DATA_BLOCK "DB_CrossCut_Opt_HMI"
{ DB_Accessible_From_OPC_UA := 'FALSE' ;
 DB_Accessible_From_Webserver := 'FALSE' ;
 S7_Optimized_Access := 'FALSE' }
VERSION : 0.1
NON_RETAIN
   STRUCT
      tALM { ExternalWritable := 'False'} : Struct   // HMI Alarms
         tE { ExternalWritable := 'False'} : Struct   // Stopping faults
            xSpare_0 { ExternalWritable := 'False'} : Bool;
            xSpare_1 { ExternalWritable := 'False'} : Bool;
            xSpare_2 { ExternalWritable := 'False'} : Bool;
            xSpare_3 { ExternalWritable := 'False'} : Bool;
            xSpare_4 { ExternalWritable := 'False'} : Bool;
            xSpare_5 { ExternalWritable := 'False'} : Bool;
            xSpare_6 { ExternalWritable := 'False'} : Bool;
            xSpare_7 { ExternalWritable := 'False'} : Bool;
            xSpare_8 { ExternalWritable := 'False'} : Bool;
            xSpare_9 { ExternalWritable := 'False'} : Bool;
            xSpare_10 { ExternalWritable := 'False'} : Bool;
            xSpare_11 { ExternalWritable := 'False'} : Bool;
            xSpare_12 { ExternalWritable := 'False'} : Bool;
            xSpare_13 { ExternalWritable := 'False'} : Bool;
            xSpare_14 { ExternalWritable := 'False'} : Bool;
            xSpare_15 { ExternalWritable := 'False'} : Bool;
            xSpare_16 { ExternalWritable := 'False'} : Bool;
            xSpare_17 { ExternalWritable := 'False'} : Bool;
            xSpare_18 { ExternalWritable := 'False'} : Bool;
            xSpare_19 { ExternalWritable := 'False'} : Bool;
            xSpare_20 { ExternalWritable := 'False'} : Bool;
            xSpare_21 { ExternalWritable := 'False'} : Bool;
            xSpare_22 { ExternalWritable := 'False'} : Bool;
            xSpare_23 { ExternalWritable := 'False'} : Bool;
            xSpare_24 { ExternalWritable := 'False'} : Bool;
            xSpare_25 { ExternalWritable := 'False'} : Bool;
            xSpare_26 { ExternalWritable := 'False'} : Bool;
            xSpare_27 { ExternalWritable := 'False'} : Bool;
            xSpare_28 { ExternalWritable := 'False'} : Bool;
            xSpare_29 { ExternalWritable := 'False'} : Bool;
            xSpare_30 { ExternalWritable := 'False'} : Bool;
            xSpare_31 { ExternalWritable := 'False'} : Bool;
         END_STRUCT;
         tS { ExternalWritable := 'False'} : Struct   // Stopping faults
            xSpare_0 { ExternalWritable := 'False'} : Bool;
            xSpare_1 { ExternalWritable := 'False'} : Bool;
            xSpare_2 { ExternalWritable := 'False'} : Bool;
            xSpare_3 { ExternalWritable := 'False'} : Bool;
            xSpare_4 { ExternalWritable := 'False'} : Bool;
            xSpare_5 { ExternalWritable := 'False'} : Bool;
            xSpare_6 { ExternalWritable := 'False'} : Bool;
            xSpare_7 { ExternalWritable := 'False'} : Bool;
            xSpare_8 { ExternalWritable := 'False'} : Bool;
            xSpare_9 { ExternalWritable := 'False'} : Bool;
            xSpare_10 { ExternalWritable := 'False'} : Bool;
            xSpare_11 { ExternalWritable := 'False'} : Bool;
            xSpare_12 { ExternalWritable := 'False'} : Bool;
            xSpare_13 { ExternalWritable := 'False'} : Bool;
            xSpare_14 { ExternalWritable := 'False'} : Bool;
            xSpare_15 { ExternalWritable := 'False'} : Bool;
            xSpare_16 { ExternalWritable := 'False'} : Bool;
            xSpare_17 { ExternalWritable := 'False'} : Bool;
            xSpare_18 { ExternalWritable := 'False'} : Bool;
            xSpare_19 { ExternalWritable := 'False'} : Bool;
            xSpare_20 { ExternalWritable := 'False'} : Bool;
            xSpare_21 { ExternalWritable := 'False'} : Bool;
            xSpare_22 { ExternalWritable := 'False'} : Bool;
            xSpare_23 { ExternalWritable := 'False'} : Bool;
            xSpare_24 { ExternalWritable := 'False'} : Bool;
            xSpare_25 { ExternalWritable := 'False'} : Bool;
            xSpare_26 { ExternalWritable := 'False'} : Bool;
            xSpare_27 { ExternalWritable := 'False'} : Bool;
            xSpare_28 { ExternalWritable := 'False'} : Bool;
            xSpare_29 { ExternalWritable := 'False'} : Bool;
            xSpare_30 { ExternalWritable := 'False'} : Bool;
            xSpare_31 { ExternalWritable := 'False'} : Bool;
         END_STRUCT;
         tF { ExternalWritable := 'False'} : Struct   // Faults
            xSpare_0 { ExternalWritable := 'False'} : Bool;
            xSpare_1 { ExternalWritable := 'False'} : Bool;
            xSpare_2 { ExternalWritable := 'False'} : Bool;
            xSpare_3 { ExternalWritable := 'False'} : Bool;
            xSpare_4 { ExternalWritable := 'False'} : Bool;
            xSpare_5 { ExternalWritable := 'False'} : Bool;
            xSpare_6 { ExternalWritable := 'False'} : Bool;
            xSpare_7 { ExternalWritable := 'False'} : Bool;
            xSpare_8 { ExternalWritable := 'False'} : Bool;
            xSpare_9 { ExternalWritable := 'False'} : Bool;
            xSpare_10 { ExternalWritable := 'False'} : Bool;
            xSpare_11 { ExternalWritable := 'False'} : Bool;
            xSpare_12 { ExternalWritable := 'False'} : Bool;
            xSpare_13 { ExternalWritable := 'False'} : Bool;
            xSpare_14 { ExternalWritable := 'False'} : Bool;
            xSpare_15 { ExternalWritable := 'False'} : Bool;
            xSpare_16 { ExternalWritable := 'False'} : Bool;
            xSpare_17 { ExternalWritable := 'False'} : Bool;
            xSpare_18 { ExternalWritable := 'False'} : Bool;
            xSpare_19 { ExternalWritable := 'False'} : Bool;
            xSpare_20 { ExternalWritable := 'False'} : Bool;
            xSpare_21 { ExternalWritable := 'False'} : Bool;
            xSpare_22 { ExternalWritable := 'False'} : Bool;
            xSpare_23 { ExternalWritable := 'False'} : Bool;
            xSpare_24 { ExternalWritable := 'False'} : Bool;
            xSpare_25 { ExternalWritable := 'False'} : Bool;
            xSpare_26 { ExternalWritable := 'False'} : Bool;
            xSpare_27 { ExternalWritable := 'False'} : Bool;
            xSpare_28 { ExternalWritable := 'False'} : Bool;
            xSpare_29 { ExternalWritable := 'False'} : Bool;
            xSpare_30 { ExternalWritable := 'False'} : Bool;
            xSpare_31 { ExternalWritable := 'False'} : Bool;
         END_STRUCT;
         tW { ExternalWritable := 'False'} : Struct   // Warnings
            xSpare_0 { ExternalWritable := 'False'} : Bool;
            xSpare_1 { ExternalWritable := 'False'} : Bool;
            xSpare_2 { ExternalWritable := 'False'} : Bool;
            xSpare_3 { ExternalWritable := 'False'} : Bool;
            xSpare_4 { ExternalWritable := 'False'} : Bool;
            xSpare_5 { ExternalWritable := 'False'} : Bool;
            xSpare_6 { ExternalWritable := 'False'} : Bool;
            xSpare_7 { ExternalWritable := 'False'} : Bool;
            xSpare_8 { ExternalWritable := 'False'} : Bool;
            xSpare_9 { ExternalWritable := 'False'} : Bool;
            xSpare_10 { ExternalWritable := 'False'} : Bool;
            xSpare_11 { ExternalWritable := 'False'} : Bool;
            xSpare_12 { ExternalWritable := 'False'} : Bool;
            xSpare_13 { ExternalWritable := 'False'} : Bool;
            xSpare_14 { ExternalWritable := 'False'} : Bool;
            xSpare_15 { ExternalWritable := 'False'} : Bool;
            xSpare_16 { ExternalWritable := 'False'} : Bool;
            xSpare_17 { ExternalWritable := 'False'} : Bool;
            xSpare_18 { ExternalWritable := 'False'} : Bool;
            xSpare_19 { ExternalWritable := 'False'} : Bool;
            xSpare_20 { ExternalWritable := 'False'} : Bool;
            xSpare_21 { ExternalWritable := 'False'} : Bool;
            xSpare_22 { ExternalWritable := 'False'} : Bool;
            xSpare_23 { ExternalWritable := 'False'} : Bool;
            xSpare_24 { ExternalWritable := 'False'} : Bool;
            xSpare_25 { ExternalWritable := 'False'} : Bool;
            xSpare_26 { ExternalWritable := 'False'} : Bool;
            xSpare_27 { ExternalWritable := 'False'} : Bool;
            xSpare_28 { ExternalWritable := 'False'} : Bool;
            xSpare_29 { ExternalWritable := 'False'} : Bool;
            xSpare_30 { ExternalWritable := 'False'} : Bool;
            xSpare_31 { ExternalWritable := 'False'} : Bool;
         END_STRUCT;
      END_STRUCT;
      tHMR { ExternalWritable := 'False'} : Struct   // HMI Read
         xEnabledPriority { ExternalWritable := 'False'} : Bool;   // Enabled/disable priority (1=enabled) {X|X|X|X|O}
         xSpare1 { ExternalWritable := 'False'} : Bool;
         xSpare2 { ExternalWritable := 'False'} : Bool;
         xSpare3 { ExternalWritable := 'False'} : Bool;
         xSpare4 { ExternalWritable := 'False'} : Bool;
         xSpare5 { ExternalWritable := 'False'} : Bool;
         xSpare6 { ExternalWritable := 'False'} : Bool;
         xSpare7 { ExternalWritable := 'False'} : Bool;
         xSpare8 { ExternalWritable := 'False'} : Bool;
         xSpare9 { ExternalWritable := 'False'} : Bool;
         xSpare10 { ExternalWritable := 'False'} : Bool;
         xSpare11 { ExternalWritable := 'False'} : Bool;
         xSpare12 { ExternalWritable := 'False'} : Bool;
         xSpare13 { ExternalWritable := 'False'} : Bool;
         xSpare14 { ExternalWritable := 'False'} : Bool;   //
         xSpare15 { ExternalWritable := 'False'} : Bool;
         xSpare16 { ExternalWritable := 'False'} : Bool;
         xSpare17 { ExternalWritable := 'False'} : Bool;
         xSpare18 { ExternalWritable := 'False'} : Bool;
         xSpare19 { ExternalWritable := 'False'} : Bool;
         xSpare20 { ExternalWritable := 'False'} : Bool;
         xSpare21 { ExternalWritable := 'False'} : Bool;
         xSpare22 { ExternalWritable := 'False'} : Bool;
         xSpare23 { ExternalWritable := 'False'} : Bool;
         xSpare24 { ExternalWritable := 'False'} : Bool;
         xSpare25 { ExternalWritable := 'False'} : Bool;
         xSpare26 { ExternalWritable := 'False'} : Bool;
         xSpare27 { ExternalWritable := 'False'} : Bool;
         xSpare28 { ExternalWritable := 'False'} : Bool;
         xSpare29 { ExternalWritable := 'False'} : Bool;
         xSpare30 { ExternalWritable := 'False'} : Bool;
         xSpare31 { ExternalWritable := 'False'} : Bool;
         xSpare { ExternalWritable := 'False'} : Array[0..15] of Bool;
         iSpare0 { ExternalWritable := 'False'} : Int;
         iSpare1 { ExternalWritable := 'False'} : Int;
         iSpare2 { ExternalWritable := 'False'} : Int;
         iSpare3 { ExternalWritable := 'False'} : Int;
         iSpare4 { ExternalWritable := 'False'} : Int;
         iSpare5 { ExternalWritable := 'False'} : Int;
         iSpare6 { ExternalWritable := 'False'} : Int;
         iSpare7 { ExternalWritable := 'False'} : Int;
         iSpare8 { ExternalWritable := 'False'} : Int;
         iSpare9 { ExternalWritable := 'False'} : Int;
         iSpare10 { ExternalWritable := 'False'} : Int;
         iSpare11 { ExternalWritable := 'False'} : Int;
         iSpare12 { ExternalWritable := 'False'} : Int;
         iSpare13 { ExternalWritable := 'False'} : Int;
         iSpare14 { ExternalWritable := 'False'} : Int;
         iSpare15 { ExternalWritable := 'False'} : Int;
         iSpare16 { ExternalWritable := 'False'} : Int;
         dSpare0 { ExternalWritable := 'False'} : DInt;   //
         dSpare1 { ExternalWritable := 'False'} : DInt;   //
         dSpare2 { ExternalWritable := 'False'} : DInt;
         dSpare3 { ExternalWritable := 'False'} : DInt;
         dSpare4 { ExternalWritable := 'False'} : DInt;
         dSpare5 { ExternalWritable := 'False'} : DInt;
         dSpare6 { ExternalWritable := 'False'} : DInt;
         dSpare7 { ExternalWritable := 'False'} : DInt;
         dSpare8 { ExternalWritable := 'False'} : DInt;
         dSpare9 { ExternalWritable := 'False'} : DInt;
         dSpare10 { ExternalWritable := 'False'} : DInt;
         dSpare11 { ExternalWritable := 'False'} : DInt;
         dSpare12 { ExternalWritable := 'False'} : DInt;
         dSpare13 { ExternalWritable := 'False'} : DInt;
         dSpare14 { ExternalWritable := 'False'} : DInt;
         dSpare15 { ExternalWritable := 'False'} : DInt;
         rSpare0 { ExternalWritable := 'False'} : Real;
         rSpare1 { ExternalWritable := 'False'} : Real;
         rSpare2 { ExternalWritable := 'False'} : Real;
         rSpare3 { ExternalWritable := 'False'} : Real;
         rSpare4 { ExternalWritable := 'False'} : Real;
         rSpare5 { ExternalWritable := 'False'} : Real;
         rSpare6 { ExternalWritable := 'False'} : Real;
         rSpare7 { ExternalWritable := 'False'} : Real;
         rSpare8 { ExternalWritable := 'False'} : Real;
         tManCmd { ExternalWritable := 'False'} : Struct
            xSpare0 { ExternalWritable := 'False'} : Bool;   //
            xSpare1 { ExternalWritable := 'False'} : Bool;
            xSpare2 { ExternalWritable := 'False'} : Bool;
            xSpare3 { ExternalWritable := 'False'} : Bool;
            xSpare4 { ExternalWritable := 'False'} : Bool;
            xSpare5 { ExternalWritable := 'False'} : Bool;
            xSpare6 { ExternalWritable := 'False'} : Bool;
            xSpare7 { ExternalWritable := 'False'} : Bool;
            xSpare8 { ExternalWritable := 'False'} : Bool;
            xSpare9 { ExternalWritable := 'False'} : Bool;
            xSpare10 { ExternalWritable := 'False'} : Bool;
            xSpare11 { ExternalWritable := 'False'} : Bool;
            xSpare12 { ExternalWritable := 'False'} : Bool;
            xSpare13 { ExternalWritable := 'False'} : Bool;
            xSpare14 { ExternalWritable := 'False'} : Bool;
            xSpare15 { ExternalWritable := 'False'} : Bool;
            xSpare { ExternalWritable := 'False'} : Array[0..15] of Bool;
         END_STRUCT;
      END_STRUCT;
      tHMW : Struct   // HMI Write
         xEnDisPriority : Bool;   // Enable/disable priority (1=enabled) {X|X|X|X|O}
         xSpare1 : Bool;
         xSpare2 : Bool;
         xSpare3 : Bool;
         xSpare4 : Bool;
         xSpare5 : Bool;
         xSpare6 : Bool;
         xSpare7 : Bool;
         xSpare8 : Bool;
         xSpare9 : Bool;
         xSpare10 : Bool;   //
         xSpare11 : Bool;
         xSpare12 : Bool;
         xSpare13 : Bool;
         xSpare14 : Bool;   //
         xSpare15 : Bool;
         xSpare16 : Bool;
         xSpare17 : Bool;
         xSpare18 : Bool;
         xSpare19 : Bool;
         xSpare20 : Bool;
         xSpare21 : Bool;
         xSpare22 : Bool;
         xSpare23 : Bool;
         xSpare24 : Bool;
         xSpare25 : Bool;
         xSpare26 : Bool;
         xSpare27 : Bool;
         xSpare28 : Bool;
         xSpare29 : Bool;
         xSpare30 : Bool;
         xSpare31 : Bool;
         xSpare : Array[0..15] of Bool;
         iSpare0 : Int;
         iSpare1 : Int;
         iSpare2 : Int;
         iSpare3 : Int;
         iSpare4 : Int;
         iSpare5 : Int;
         iSpare6 : Int;
         iSpare7 : Int;
         iSpare8 : Int;
         iSpare9 : Int;
         iSpare10 : Int;
         iSpare11 : Int;
         iSpare12 : Int;
         iSpare13 : Int;
         iSpare14 : Int;
         iSpare15 : Int;
         iSpare16 : Int;
         dSpare0 : DInt;   //
         dSpare1 : Int;   //
         dSpare2 : Int;   //
         dSpare3 : DInt;
         dSpare4 : DInt;
         dSpare5 : DInt;
         dSpare6 : DInt;
         dSpare7 : DInt;
         dSpare8 : DInt;
         dSpare9 : DInt;
         dSpare10 : DInt;
         dSpare11 : DInt;
         dSpare12 : DInt;
         dSpare13 : DInt;
         dSpare14 : DInt;
         dSpare15 : DInt;
         dSpare16 : DInt;
         rSpare0 : Real;
         rSpare1 : Real;
         rSpare2 : Real;
         rSpare3 : Real;
         rSpare4 : Real;
         rSpare5 : Real;
         rSpare6 : Real;
         rSpare7 : Real;
         rSpare8 : Real;
         tManCmd : Struct
            xSpare0 : Bool;   //
            xSpare1 : Bool;
            xSpare2 { ExternalWritable := 'False'} : Bool;
            xSpare3 { ExternalWritable := 'False'} : Bool;
            xSpare4 { ExternalWritable := 'False'} : Bool;
            xSpare5 { ExternalWritable := 'False'} : Bool;
            xSpare6 { ExternalWritable := 'False'} : Bool;
            xSpare7 { ExternalWritable := 'False'} : Bool;
            xSpare8 { ExternalWritable := 'False'} : Bool;
            xSpare9 { ExternalWritable := 'False'} : Bool;
            xSpare10 { ExternalWritable := 'False'} : Bool;
            xSpare11 { ExternalWritable := 'False'} : Bool;
            xSpare12 { ExternalWritable := 'False'} : Bool;
            xSpare13 { ExternalWritable := 'False'} : Bool;
            xSpare14 { ExternalWritable := 'False'} : Bool;
            xSpare15 { ExternalWritable := 'False'} : Bool;
            xSpare16 : Bool;
            xSpare17 : Bool;
            xSpare18 : Bool;
            xSpare19 : Bool;
            xSpare20 : Bool;
            xSpare21 : Bool;
            xSpare22 : Bool;
            xSpare23 : Bool;
            xSpare24 : Bool;
            xSpare25 : Bool;
            xSpare26 : Bool;
            xSpare27 : Bool;
            xSpare28 : Bool;
            xSpare29 : Bool;
            xSpare30 : Bool;
            xSpare31 : Bool;
         END_STRUCT;
      END_STRUCT;
   END_STRUCT;


BEGIN

END_DATA_BLOCK

DATA_BLOCK "DB_CrossCut_1_HMI"
{ DB_Accessible_From_OPC_UA := 'FALSE' ;
 DB_Accessible_From_Webserver := 'FALSE' ;
 S7_Optimized_Access := 'FALSE' }
VERSION : 0.1
NON_RETAIN
   STRUCT
      tALM : Struct   // HMI Alarms
         tE : Struct   // Emergency alarms
            xLocON : Bool;   // KE.Local emergency ON {X|X|X|X|O}
            xLocal1 : Bool;   // SB.Local emergency push button 1 {X|X|X|X|O}
            xLocal2 : Bool;   // SB.Local emergency push button 2 {X|X|X|X|O}
            xLocal3 : Bool;   // SB.Local emergency push button 3 {X|X|X|X|O}
            xSpare_4 : Bool;
            xSpare_5 : Bool;
            xSpare_6 : Bool;
            xSpare_7 : Bool;
            xSpare_8 : Bool;
            xSpare_9 : Bool;
            xSpare_10 : Bool;
            xSpare_11 : Bool;
            xSpare_12 : Bool;
            xSpare_13 : Bool;
            xSpare_14 : Bool;
            xSpare_15 : Bool;
            xSpare_16 : Bool;
            xSpare_17 : Bool;
            xSpare_18 : Bool;
            xSpare_19 : Bool;
            xSpare_20 : Bool;
            xSpare_21 : Bool;
            xSpare_22 : Bool;
            xSpare_23 : Bool;
            xSpare_24 : Bool;
            xSpare_25 : Bool;
            xSpare_26 : Bool;
            xSpare_27 : Bool;
            xSpare_28 : Bool;
            xSpare_29 : Bool;
            xSpare_30 : Bool;
            xSpare_31 : Bool;
         END_STRUCT;
         tS : Struct   // Stopping faults
            xAxisNotAvail : Bool;   // AZ.Axis not available {X|X|X|X|O}
            xInpInstallation : Bool;   // L+.Input power supply ON {X|X|X|X|O}
            xAuxPower : Bool;   // L+.Auxiliary power supple set-in {X|X|X|X|O}
            xAreaSafety : Bool;   // KE.Area safety {X|X|X|X|O}
            xOverstroke : Bool;   // KA.Carriage overstroke {X|X|X|X|O}
            xExternInputPower : Bool;   // L+.External input power supply {X|X|X|X|O}
            xCarriageCutOut : Bool;   // QM.Carriage translation overload {X|X|X|X|O}
            xDriveTrip : Bool;   // AZ.Drive trip {X|X|X|X|O}
            xDriveNotEnabled : Bool;   // AZ.Drive not enabled {X|X|X|X|O}
            xAxisNotReady : Bool;   // AZ.Axis not ready {X|X|X|X|O}
            xDriveNotReady : Bool;   // AZ.Drive not ready {X|X|X|X|O}
            xAxisNotSyncro : Bool;   // AZ.Axis not syncronized {X|X|X|X|O}
            xSpare_12 : Bool;
            xSpare_13 : Bool;
            xSpare_14 : Bool;
            xSpare_15 : Bool;
            xSpare_16 : Bool;
            xSpare_17 : Bool;
            xSpare_18 : Bool;
            xSpare_19 : Bool;
            xSpare_20 : Bool;
            xSpare_21 : Bool;
            xSpare_22 : Bool;
            xSpare_23 : Bool;
            xSpare_24 : Bool;
            xSpare_25 : Bool;
            xSpare_26 : Bool;
            xSpare_27 : Bool;
            xSpare_28 : Bool;
            xSpare_29 : Bool;
            xSpare_30 : Bool;
            xSpare_31 : Bool;
         END_STRUCT;
         tF : Struct   // Faults
            xSpare_0 : Bool;
            xSpare_1 : Bool;
            xSpare_2 : Bool;
            xSpare_3 : Bool;
            xSpare_4 : Bool;
            xSpare_5 : Bool;
            xSpare_6 : Bool;
            xSpare_7 : Bool;
            xSpare_8 : Bool;
            xSpare_9 : Bool;
            xSpare_10 : Bool;
            xSpare_11 : Bool;
            xSpare_12 : Bool;
            xSpare_13 : Bool;
            xSpare_14 : Bool;
            xSpare_15 : Bool;
            xSpare_16 : Bool;
            xSpare_17 : Bool;
            xSpare_18 : Bool;
            xSpare_19 : Bool;
            xSpare_20 : Bool;
            xSpare_21 : Bool;
            xSpare_22 : Bool;
            xSpare_23 : Bool;
            xSpare_24 : Bool;
            xSpare_25 : Bool;
            xSpare_26 : Bool;
            xSpare_27 : Bool;
            xSpare_28 : Bool;
            xSpare_29 : Bool;
            xSpare_30 : Bool;
            xSpare_31 : Bool;
         END_STRUCT;
         tW : Struct   // Warnings
            xSpare_0 : Bool;
            xSpare_1 : Bool;
            xSpare_2 : Bool;
            xSpare_3 : Bool;
            xSpare_4 : Bool;
            xSpare_5 : Bool;
            xSpare_6 : Bool;
            xSpare_7 : Bool;
            xSpare_8 : Bool;
            xSpare_9 : Bool;
            xSpare_10 : Bool;
            xSpare_11 : Bool;
            xSpare_12 : Bool;
            xSpare_13 : Bool;
            xSpare_14 : Bool;
            xSpare_15 : Bool;
            xSpare_16 : Bool;
            xSpare_17 : Bool;
            xSpare_18 : Bool;
            xSpare_19 : Bool;
            xSpare_20 : Bool;
            xSpare_21 : Bool;
            xSpare_22 : Bool;
            xSpare_23 : Bool;
            xSpare_24 : Bool;
            xSpare_25 : Bool;
            xSpare_26 : Bool;
            xSpare_27 : Bool;
            xSpare_28 : Bool;
            xSpare_29 : Bool;
            xSpare_30 : Bool;
            xSpare_31 : Bool;
         END_STRUCT;
      END_STRUCT;
      tHMR : Struct   // HMI Read
         xSpare0 : Bool;   //
         xSpare1 : Bool;   //
         xSpare2 : Bool;
         xSpare3 : Bool;
         xSpare4 : Bool;
         xSpare5 : Bool;
         xSpare6 : Bool;
         xSpare7 : Bool;
         xSpare8 : Bool;
         xSpare9 : Bool;
         xSpare10 : Bool;
         xSpare11 : Bool;
         xSpare12 : Bool;
         xSpare13 : Bool;
         xManualCommandEnabled : Bool;   // Manual Command enabled {x|x|x|x|O}
         xSpare15 : Bool;
         xSpare16 : Bool;
         xSpare17 : Bool;
         xSpare18 : Bool;
         xSpare19 : Bool;
         xSpare20 : Bool;
         xSpare21 : Bool;
         xSpare22 : Bool;
         xSpare23 : Bool;
         xSpare24 : Bool;
         xSpare25 : Bool;
         xSpare26 : Bool;
         xSpare27 : Bool;
         xSpare28 : Bool;
         xSpare29 : Bool;
         xSpare30 : Bool;
         xSpare31 : Bool;
         xSpare : Array[0..15] of Bool;
         iSpare0 { ExternalWritable := 'False'} : Int;
         iSpare1 { ExternalWritable := 'False'} : Int;
         iSpare2 { ExternalWritable := 'False'} : Int;
         iSpare3 { ExternalWritable := 'False'} : Int;
         iSpare4 { ExternalWritable := 'False'} : Int;
         iSpare5 { ExternalWritable := 'False'} : Int;
         iSpare6 { ExternalWritable := 'False'} : Int;
         iSpare7 { ExternalWritable := 'False'} : Int;
         iSpare8 { ExternalWritable := 'False'} : Int;
         iSpare9 { ExternalWritable := 'False'} : Int;
         iSpare10 { ExternalWritable := 'False'} : Int;
         iSpare11 { ExternalWritable := 'False'} : Int;
         iSpare12 { ExternalWritable := 'False'} : Int;
         iSpare13 { ExternalWritable := 'False'} : Int;
         iSpare14 { ExternalWritable := 'False'} : Int;
         iSpare15 { ExternalWritable := 'False'} : Int;
         iSpare16 { ExternalWritable := 'False'} : Int;
         dDistanceSnaproll_cmm { ExternalWritable := 'False'} : DInt;   // Distance from snaproll [mm/100] {mm/100|mm|x|x|M}
         dStatus { ExternalWritable := 'False'} : DInt;   // XCut actual status (1=Idle 3=Running 7=Faulted)  {X|X|X|X|O}
         dXCutActualStatus { ExternalWritable := 'False'} : DInt;   // XCut actual status (1=Disabled 3=Enabled) {X|X|X|X|O}
         dXCutStatusRequest { ExternalWritable := 'False'} : DInt;   // XCut status request (1=Disabled 3=Enabled) {X|X|X|X|O}
         dDistanceFromCenterLine_cmm { ExternalWritable := 'False'} : DInt;   // Distance from center line [mm/100] {mm/100|mm|X|X|O}
         dAngleValue_uDegree { ExternalWritable := 'False'} : DInt;   // Angle value [°/1000000] {°/1000000|°|X|X|O}
         dActualCutPosRequest { ExternalWritable := 'False'} : DInt;   // Actual cut position request (1=By operator 2=On gross ribbon 3=On net ribbon 4=On YCut position) {X|X|X|X|O}
         dCarriagePosition_cmm { ExternalWritable := 'False'} : DInt;   // Actual carriage position [mm/100]
         dSpare8 { ExternalWritable := 'False'} : DInt;
         dSpare9 { ExternalWritable := 'False'} : DInt;
         dSpare10 { ExternalWritable := 'False'} : DInt;
         dSpare11 { ExternalWritable := 'False'} : DInt;
         dSpare12 { ExternalWritable := 'False'} : DInt;
         dSpare13 { ExternalWritable := 'False'} : DInt;
         dSpare14 { ExternalWritable := 'False'} : DInt;
         dSpare15 { ExternalWritable := 'False'} : DInt;
         rHeadUsage_km { ExternalWritable := 'False'} : Real;   // Head usage [Km] {Km|Km|X|X|O}
         rSpare1 { ExternalWritable := 'False'} : Real;
         rSpare2 { ExternalWritable := 'False'} : Real;
         rSpare3 { ExternalWritable := 'False'} : Real;
         rSpare4 { ExternalWritable := 'False'} : Real;
         rSpare5 { ExternalWritable := 'False'} : Real;
         rSpare6 { ExternalWritable := 'False'} : Real;
         rSpare7 { ExternalWritable := 'False'} : Real;
         rSpare8 { ExternalWritable := 'False'} : Real;
         tManCmd { ExternalWritable := 'False'} : Struct
            xManJogFwdFdbk { ExternalWritable := 'False'} : Bool;   // Manual jog forward feedback {X|X|X|X|O}
            xManJogBckFdbk { ExternalWritable := 'False'} : Bool;   // Manual jog backward feedback {X|X|X|X|O}
            xManCarriageDownFdbk { ExternalWritable := 'False'} : Bool;   // Manual carriage down feedback {X|X|X|X|O}
            xManFireONFdbk { ExternalWritable := 'False'} : Bool;   // Manual fire ON feedback {X|X|X|X|O}
            xManOilONFdbk { ExternalWritable := 'False'} : Bool;   // Manual oil ON feedback {X|X|X|X|O}
            xSpare5 { ExternalWritable := 'False'} : Bool;
            xSpare6 { ExternalWritable := 'False'} : Bool;
            xSpare7 { ExternalWritable := 'False'} : Bool;
            xSpare8 { ExternalWritable := 'False'} : Bool;
            xSpare9 { ExternalWritable := 'False'} : Bool;
            xSpare10 { ExternalWritable := 'False'} : Bool;
            xSpare11 { ExternalWritable := 'False'} : Bool;
            xSpare12 { ExternalWritable := 'False'} : Bool;
            xSpare13 { ExternalWritable := 'False'} : Bool;
            xSpare14 { ExternalWritable := 'False'} : Bool;
            xSpare15 { ExternalWritable := 'False'} : Bool;
            xSpare { ExternalWritable := 'False'} : Array[0..15] of Bool;
         END_STRUCT;
      END_STRUCT;
      tHMW : Struct   // HMI Write
         xCutBreakEnabled { ExternalWritable := 'False'} : Bool;   // Cut on glass break enabled {X|X|X|X|O}
         xIncAngleValue : Bool;   // Increment angle value {X|X|X|X|O}
         xDecAngleValue : Bool;   // Decrement angle value {X|X|X|X|O}
         xCalibDistRequest : Bool;   // Calibration distance request {X|X|X|X|O}
         xCalibDiagRequest : Bool;   // Calibration diagonal request {X|X|X|X|O}
         xCutOperator : Bool;   // Cutting position by operator request {X|X|X|X|O}
         xCutGross : Bool;   // Cutting position by gross width position {X|X|X|X|O}
         xCutNet : Bool;   // Cutting position by net width position {X|X|X|X|O}
         xCutYCut : Bool;   // Cutting position by YCut position {X|X|X|X|O}
         xSpare9 : Bool;
         xSpare10 : Bool;
         xSpare11 : Bool;
         xSpare12 : Bool;
         xResetHeadUsage : Bool;   // Reset the head usage {X|X|X|X|O}
         xEnableManualCommand : Bool;   // Enable Disable Manual command {x|x|x|x|O}
         xUpdateDistanceSnaproll : Bool;   // Update distance from snaproll {x|x|x|x|M}
         xUpdateDistCenterLine : Bool;   // Update distance from center line {X|X|X|X|M}
         xUpdateAngleValue : Bool;   // Update angle value {X|X|X|X|M}
         xSpare18 : Bool;
         xSpare19 : Bool;
         xSpare20 : Bool;
         xSpare21 : Bool;
         xSpare22 : Bool;
         xSpare23 : Bool;
         xSpare24 : Bool;
         xSpare25 : Bool;
         xSpare26 : Bool;
         xSpare27 : Bool;
         xSpare28 : Bool;
         xSpare29 : Bool;
         xSpare30 : Bool;
         xSpare31 : Bool;
         xSpare : Array[0..15] of Bool;
         iSpare0 : Int;
         iSpare1 : Int;
         iSpare2 : Int;
         iSpare3 : Int;
         iSpare4 : Int;
         iSpare5 : Int;
         iSpare6 : Int;
         iSpare7 : Int;
         iSpare8 : Int;
         iSpare9 : Int;
         iSpare10 : Int;
         iSpare11 : Int;
         iSpare12 : Int;
         iSpare13 : Int;
         iSpare14 : Int;
         iSpare15 : Int;
         iSpare16 : Int;
         dDistanceSnaproll_cmm : DInt;   // Distance from snaproll [mm/100] {mm/100|mm|1|70000|M}
         dDistanceFromCenterLine_cmm : DInt;   // Distance from center line [mm/100] {mm/100|mm|-3000|0|M}
         dAngleValue_uDegree : DInt;   // Bridge angle value [°/1000000] {°/1000000|°|7|9|M}
         dOperStartCutPos_cmm : DInt;   // Operator start cut position [mm/100] {mm/100|mm|-3000|0|O}
         dOperEndCutPos_cmm : DInt;   // Operator end cut position  [mm/100] {mm/100|mm|0|3000|O}
         dDescReactTime_ms : DInt;   // Carriage descent reaction time [ms] {ms|s|0|1|M}
         dRaiseReactTime_ms : DInt;   // Carriage raise reaction time [ms] {ms|s|0|1|M}
         dFireONReactTime_ms : DInt;   // Fire ON reaction time [ms] {ms|s|0|1|M}
         dFireOFFReactTime_ms : DInt;   // Fire OFF reaction time [ms] {ms|s|0|1|M}
         dOilONDelay_ms : DInt;   // Oil ON delay [ms] {ms|s|-1|1|O}
         dOilOFFDelay_ms : DInt;   // Oil OFF delay [ms] {ms|s|-1|1|O}
         dCutStartOffsetDelay_cmm : DInt;   // Start cut offset delay [mm/100] {mm/100|mm|-500|500|O}
         dCutEndOffsetDelay_cmm : DInt;   // End cut offset delay [mm/100] {mm/100|mm|-500|500|O}
         dDistTeoLength_cmm : DInt;   // Calibration distance.Theorical length [mm/100] {mm/100|mm|0|7000|O}
         dDistRealLength_cmm : DInt;   // Calibration distance.Real length [mm/100] {mm/100|mm|0|7000|O}
         dDiagRealLength_cmm : DInt;   // Calibration diagonal.Real length [mm/100] {mm/100|mm|0|7000|O}
         dDiagRealWidth_cmm : DInt;   // Calibration diagonal.Real width [mm/100] {mm/100|mm|0|4000|O}
         dDiagGlassFlow_cmm : DInt;   // Calibration diagonal.Real length diagonal glass flow [mm/100] {mm/100|mm|0|10000|O}
         dDiagGlassOppFlow_cmm : DInt;   // Calibration diagonal.Real length diagonal opposite glass flow [mm/100] {mm/100|mm|0|10000|O}
         dCuttingPressure_mN : DInt;   // Cutting pressure [N/1000] {N/1000|N|9|180|O}
         dPosOffset_cmm : DInt;   // Calibration offset distance from snaproll [mm/100]  {mm/100|mm|-50|50|O}
         dCutPriority : DInt;   // Cut priority number  {X|X|0|5|O}
         dSpare22 : DInt;
         rSpare6 : Real;
         rSpare7 : Real;
         rSpare8 : Real;
         tManCmd : Struct
            xMan_JogForward : Bool;   // Manual mode - Jog forward {X|X|X|X|M}
            xMan_JobBackward : Bool;   // Manual mode - Jog backward {X|X|X|X|M}
            xMan_CarriageDown : Bool;   // Manual mode - Carriage down {X|X|X|X|M}
            xMan_FireOn : Bool;   // Manual mode - Fire ON {X|X|X|X|M}
            xMan_OilOn : Bool;   // Manual mode - Oil ON {X|X|X|X|M}
            xSpare5 { ExternalWritable := 'False'} : Bool;
            xSpare6 { ExternalWritable := 'False'} : Bool;
            xSpare7 { ExternalWritable := 'False'} : Bool;
            xSpare8 { ExternalWritable := 'False'} : Bool;
            xSpare9 { ExternalWritable := 'False'} : Bool;
            xSpare10 { ExternalWritable := 'False'} : Bool;
            xSpare11 { ExternalWritable := 'False'} : Bool;
            xSpare12 { ExternalWritable := 'False'} : Bool;
            xSpare13 { ExternalWritable := 'False'} : Bool;
            xSpare14 { ExternalWritable := 'False'} : Bool;
            xSpare15 { ExternalWritable := 'False'} : Bool;
            xSpare16 : Bool;
            xSpare17 : Bool;
            xSpare18 : Bool;
            xSpare19 : Bool;
            xSpare20 : Bool;
            xSpare21 : Bool;
            xSpare22 : Bool;
            xSpare23 : Bool;
            xSpare24 : Bool;
            xSpare25 : Bool;
            xSpare26 : Bool;
            xSpare27 : Bool;
            xSpare28 : Bool;
            xSpare29 : Bool;
            xSpare30 : Bool;
            xSpare31 : Bool;
         END_STRUCT;
      END_STRUCT;
   END_STRUCT;


BEGIN

END_DATA_BLOCK

DATA_BLOCK "DB_Breaker_M206_HMI"
{ DB_Accessible_From_OPC_UA := 'FALSE' ;
 DB_Accessible_From_Webserver := 'FALSE' ;
 S7_Optimized_Access := 'FALSE' }
VERSION : 0.1
NON_RETAIN
   STRUCT
      tALM { ExternalWritable := 'False'} : Struct   // HMI Alarms
         tE { ExternalWritable := 'False'} : Struct   // Stopping faults
            xSpare_0 { ExternalWritable := 'False'} : Bool;
            xSpare_1 { ExternalWritable := 'False'} : Bool;
            xSpare_2 { ExternalWritable := 'False'} : Bool;
            xSpare_3 { ExternalWritable := 'False'} : Bool;
            xSpare_4 { ExternalWritable := 'False'} : Bool;
            xSpare_5 { ExternalWritable := 'False'} : Bool;
            xSpare_6 { ExternalWritable := 'False'} : Bool;
            xSpare_7 { ExternalWritable := 'False'} : Bool;
            xSpare_8 { ExternalWritable := 'False'} : Bool;
            xSpare_9 { ExternalWritable := 'False'} : Bool;
            xSpare_10 { ExternalWritable := 'False'} : Bool;
            xSpare_11 { ExternalWritable := 'False'} : Bool;
            xSpare_12 { ExternalWritable := 'False'} : Bool;
            xSpare_13 { ExternalWritable := 'False'} : Bool;
            xSpare_14 { ExternalWritable := 'False'} : Bool;
            xSpare_15 { ExternalWritable := 'False'} : Bool;
            xSpare_16 { ExternalWritable := 'False'} : Bool;
            xSpare_17 { ExternalWritable := 'False'} : Bool;
            xSpare_18 { ExternalWritable := 'False'} : Bool;
            xSpare_19 { ExternalWritable := 'False'} : Bool;
            xSpare_20 { ExternalWritable := 'False'} : Bool;
            xSpare_21 { ExternalWritable := 'False'} : Bool;
            xSpare_22 { ExternalWritable := 'False'} : Bool;
            xSpare_23 { ExternalWritable := 'False'} : Bool;
            xSpare_24 { ExternalWritable := 'False'} : Bool;
            xSpare_25 { ExternalWritable := 'False'} : Bool;
            xSpare_26 { ExternalWritable := 'False'} : Bool;
            xSpare_27 { ExternalWritable := 'False'} : Bool;
            xSpare_28 { ExternalWritable := 'False'} : Bool;
            xSpare_29 { ExternalWritable := 'False'} : Bool;
            xSpare_30 { ExternalWritable := 'False'} : Bool;
            xSpare_31 { ExternalWritable := 'False'} : Bool;
         END_STRUCT;
         tS { ExternalWritable := 'False'} : Struct   // Stopping faults machine
            xSpare_1 { ExternalWritable := 'False'} : Bool;
            xConditionOKCulletSystem { ExternalWritable := 'False'} : Bool;   // Condition OK from cullet system {X|X|X|X|O}
            xBreakerRotationFeedback { ExternalWritable := 'False'} : Bool;   // M206SQ1.Breaker rotation feedback {X|X|X|X|O}
            xBreakerKmRotationFeedback { ExternalWritable := 'False'} : Bool;
            xSpare_3 { ExternalAccessible := 'False'; ExternalVisible := 'False'; ExternalWritable := 'False'} : Bool;
            xProtectionBreakerRotation { ExternalWritable := 'False'} : Bool;   // A176QM1.Protection breaker rotation {X|X|X|X|O}
            xSpare_4 { ExternalAccessible := 'False'; ExternalVisible := 'False'; ExternalWritable := 'False'} : Bool;
            xSpare_5 { ExternalAccessible := 'False'; ExternalVisible := 'False'; ExternalWritable := 'False'} : Bool;
            xSpare_6 { ExternalAccessible := 'False'; ExternalVisible := 'False'; ExternalWritable := 'False'} : Bool;
            xSpare_7 { ExternalAccessible := 'False'; ExternalVisible := 'False'; ExternalWritable := 'False'} : Bool;
            xSpare_8 { ExternalAccessible := 'False'; ExternalVisible := 'False'; ExternalWritable := 'False'} : Bool;
            xSpare_9 { ExternalAccessible := 'False'; ExternalVisible := 'False'; ExternalWritable := 'False'} : Bool;
            xSpare_10 { ExternalAccessible := 'False'; ExternalVisible := 'False'; ExternalWritable := 'False'} : Bool;
            xSpare_11 { ExternalAccessible := 'False'; ExternalVisible := 'False'; ExternalWritable := 'False'} : Bool;
            xSpare_14 { ExternalAccessible := 'False'; ExternalVisible := 'False'; ExternalWritable := 'False'} : Bool;
            xSpare_15 { ExternalAccessible := 'False'; ExternalVisible := 'False'; ExternalWritable := 'False'} : Bool;
            xSpare_16 { ExternalAccessible := 'False'; ExternalVisible := 'False'; ExternalWritable := 'False'} : Bool;
            xSpare_17 { ExternalAccessible := 'False'; ExternalVisible := 'False'; ExternalWritable := 'False'} : Bool;
            xSpare_18 { ExternalAccessible := 'False'; ExternalVisible := 'False'; ExternalWritable := 'False'} : Bool;
            xSpare_19 { ExternalAccessible := 'False'; ExternalVisible := 'False'; ExternalWritable := 'False'} : Bool;
            xSpare_20 { ExternalAccessible := 'False'; ExternalVisible := 'False'; ExternalWritable := 'False'} : Bool;
            xSpare_21 { ExternalAccessible := 'False'; ExternalVisible := 'False'; ExternalWritable := 'False'} : Bool;
            xSpare_22 { ExternalAccessible := 'False'; ExternalVisible := 'False'; ExternalWritable := 'False'} : Bool;
            xSpare_23 { ExternalAccessible := 'False'; ExternalVisible := 'False'; ExternalWritable := 'False'} : Bool;
            xSpare_24 { ExternalAccessible := 'False'; ExternalVisible := 'False'; ExternalWritable := 'False'} : Bool;
            xSpare_25 { ExternalAccessible := 'False'; ExternalVisible := 'False'; ExternalWritable := 'False'} : Bool;
            xSpare_26 { ExternalAccessible := 'False'; ExternalVisible := 'False'; ExternalWritable := 'False'} : Bool;
            xSpare_27 { ExternalAccessible := 'False'; ExternalVisible := 'False'; ExternalWritable := 'False'} : Bool;
            xSpare_28 { ExternalAccessible := 'False'; ExternalVisible := 'False'; ExternalWritable := 'False'} : Bool;
            xSpare_29 { ExternalAccessible := 'False'; ExternalVisible := 'False'; ExternalWritable := 'False'} : Bool;
            xSpare_30 { ExternalAccessible := 'False'; ExternalVisible := 'False'; ExternalWritable := 'False'} : Bool;
            xSpare_31 { ExternalAccessible := 'False'; ExternalVisible := 'False'; ExternalWritable := 'False'} : Bool;
         END_STRUCT;
         tF { ExternalWritable := 'False'} : Struct   // Faults
            xSpare_0 { ExternalWritable := 'False'} : Bool;
            xSpare_1 { ExternalWritable := 'False'} : Bool;
            xSpare_2 { ExternalWritable := 'False'} : Bool;
            xSpare_3 { ExternalWritable := 'False'} : Bool;
            xSpare_4 { ExternalWritable := 'False'} : Bool;
            xSpare_5 { ExternalWritable := 'False'} : Bool;
            xSpare_6 { ExternalWritable := 'False'} : Bool;
            xSpare_7 { ExternalWritable := 'False'} : Bool;
            xSpare_8 { ExternalWritable := 'False'} : Bool;
            xSpare_9 { ExternalWritable := 'False'} : Bool;
            xSpare_10 { ExternalWritable := 'False'} : Bool;
            xSpare_11 { ExternalWritable := 'False'} : Bool;
            xSpare_12 { ExternalWritable := 'False'} : Bool;
            xSpare_13 { ExternalWritable := 'False'} : Bool;
            xSpare_14 { ExternalWritable := 'False'} : Bool;
            xSpare_15 { ExternalWritable := 'False'} : Bool;
            xSpare_16 { ExternalWritable := 'False'} : Bool;
            xSpare_17 { ExternalWritable := 'False'} : Bool;
            xSpare_18 { ExternalWritable := 'False'} : Bool;
            xSpare_19 { ExternalWritable := 'False'} : Bool;
            xSpare_20 { ExternalWritable := 'False'} : Bool;
            xSpare_21 { ExternalWritable := 'False'} : Bool;
            xSpare_22 { ExternalWritable := 'False'} : Bool;
            xSpare_23 { ExternalWritable := 'False'} : Bool;
            xSpare_24 { ExternalWritable := 'False'} : Bool;
            xSpare_25 { ExternalWritable := 'False'} : Bool;
            xSpare_26 { ExternalWritable := 'False'} : Bool;
            xSpare_27 { ExternalWritable := 'False'} : Bool;
            xSpare_28 { ExternalWritable := 'False'} : Bool;
            xSpare_29 { ExternalWritable := 'False'} : Bool;
            xSpare_30 { ExternalWritable := 'False'} : Bool;
            xSpare_31 { ExternalWritable := 'False'} : Bool;
         END_STRUCT;
         tW { ExternalWritable := 'False'} : Struct   // Warnings
            xSpare_0 { ExternalWritable := 'False'} : Bool;
            xSpare_1 { ExternalWritable := 'False'} : Bool;
            xSpare_2 { ExternalWritable := 'False'} : Bool;
            xSpare_3 { ExternalWritable := 'False'} : Bool;
            xSpare_4 { ExternalWritable := 'False'} : Bool;
            xSpare_5 { ExternalWritable := 'False'} : Bool;
            xSpare_6 { ExternalWritable := 'False'} : Bool;
            xSpare_7 { ExternalWritable := 'False'} : Bool;
            xSpare_8 { ExternalWritable := 'False'} : Bool;
            xSpare_9 { ExternalWritable := 'False'} : Bool;
            xSpare_10 { ExternalWritable := 'False'} : Bool;
            xSpare_11 { ExternalWritable := 'False'} : Bool;
            xSpare_12 { ExternalWritable := 'False'} : Bool;
            xSpare_13 { ExternalWritable := 'False'} : Bool;
            xSpare_14 { ExternalWritable := 'False'} : Bool;
            xSpare_15 { ExternalWritable := 'False'} : Bool;
            xSpare_16 { ExternalWritable := 'False'} : Bool;
            xSpare_17 { ExternalWritable := 'False'} : Bool;
            xSpare_18 { ExternalWritable := 'False'} : Bool;
            xSpare_19 { ExternalWritable := 'False'} : Bool;
            xSpare_20 { ExternalWritable := 'False'} : Bool;
            xSpare_21 { ExternalWritable := 'False'} : Bool;
            xSpare_22 { ExternalWritable := 'False'} : Bool;
            xSpare_23 { ExternalWritable := 'False'} : Bool;
            xSpare_24 { ExternalWritable := 'False'} : Bool;
            xSpare_25 { ExternalWritable := 'False'} : Bool;
            xSpare_26 { ExternalWritable := 'False'} : Bool;
            xSpare_27 { ExternalWritable := 'False'} : Bool;
            xSpare_28 { ExternalWritable := 'False'} : Bool;
            xSpare_29 { ExternalWritable := 'False'} : Bool;
            xSpare_30 { ExternalWritable := 'False'} : Bool;
            xSpare_31 { ExternalWritable := 'False'} : Bool;
         END_STRUCT;
      END_STRUCT;
      tHMR { ExternalWritable := 'False'} : Struct   // HMI Read
         xEnabledRunAlwaysModeBreaker { ExternalWritable := 'False'} : Bool;   // Enabled run always breaker {x|x|x|x|O}
         xSpare1 { ExternalWritable := 'False'} : Bool;
         xSpare2 { ExternalWritable := 'False'} : Bool;
         xSpare3 { ExternalWritable := 'False'} : Bool;
         xSpare4 { ExternalWritable := 'False'} : Bool;
         xSpare5 { ExternalWritable := 'False'} : Bool;
         xSpare6 { ExternalWritable := 'False'} : Bool;
         xSpare7 { ExternalWritable := 'False'} : Bool;
         xSpare8 { ExternalWritable := 'False'} : Bool;
         xSpare9 { ExternalWritable := 'False'} : Bool;
         xSpare10 { ExternalWritable := 'False'} : Bool;
         xSpare11 { ExternalWritable := 'False'} : Bool;
         xSpare12 { ExternalWritable := 'False'} : Bool;
         xSpare13 { ExternalWritable := 'False'} : Bool;
         xManualCommandEnabled { ExternalWritable := 'False'} : Bool;   // Manual Command enabled {x|x|x|x|O}
         xSpare15 { ExternalWritable := 'False'} : Bool;
         xSpare16 { ExternalWritable := 'False'} : Bool;
         xSpare17 { ExternalWritable := 'False'} : Bool;
         xSpare18 { ExternalWritable := 'False'} : Bool;
         xSpare19 { ExternalWritable := 'False'} : Bool;
         xSpare20 { ExternalWritable := 'False'} : Bool;
         xSpare21 { ExternalWritable := 'False'} : Bool;
         xSpare22 { ExternalWritable := 'False'} : Bool;
         xSpare23 { ExternalWritable := 'False'} : Bool;
         xSpare24 { ExternalWritable := 'False'} : Bool;
         xSpare25 { ExternalWritable := 'False'} : Bool;
         xSpare26 { ExternalWritable := 'False'} : Bool;
         xSpare27 { ExternalWritable := 'False'} : Bool;
         xSpare28 { ExternalWritable := 'False'} : Bool;
         xSpare29 { ExternalWritable := 'False'} : Bool;
         xSpare30 { ExternalWritable := 'False'} : Bool;
         xSpare31 { ExternalWritable := 'False'} : Bool;
         xSpare { ExternalWritable := 'False'} : Array[0..15] of Bool;
         iSpare0 { ExternalWritable := 'False'} : Int;
         iSpare1 { ExternalWritable := 'False'} : Int;
         iSpare2 { ExternalWritable := 'False'} : Int;
         iSpare3 { ExternalWritable := 'False'} : Int;
         iSpare4 { ExternalWritable := 'False'} : Int;
         iSpare5 { ExternalWritable := 'False'} : Int;
         iSpare6 { ExternalWritable := 'False'} : Int;
         iSpare7 { ExternalWritable := 'False'} : Int;
         iSpare8 { ExternalWritable := 'False'} : Int;
         iSpare9 { ExternalWritable := 'False'} : Int;
         iSpare10 { ExternalWritable := 'False'} : Int;
         iSpare11 { ExternalWritable := 'False'} : Int;
         iSpare12 { ExternalWritable := 'False'} : Int;
         iSpare13 { ExternalWritable := 'False'} : Int;
         iSpare14 { ExternalWritable := 'False'} : Int;
         iSpare15 { ExternalWritable := 'False'} : Int;
         iSpare16 { ExternalWritable := 'False'} : Int;
         dStatus { ExternalWritable := 'False'} : DInt;   // Status (1=Idle 3=Run 7=Anomaly) {X|X|X|X|O}
         dSpare1 { ExternalWritable := 'False'} : DInt;
         dSpare2 { ExternalWritable := 'False'} : DInt;
         dSpare3 { ExternalWritable := 'False'} : DInt;
         dSpare4 { ExternalWritable := 'False'} : DInt;
         dSpare5 { ExternalWritable := 'False'} : DInt;
         dSpare6 { ExternalWritable := 'False'} : DInt;
         dSpare7 { ExternalWritable := 'False'} : DInt;
         dSpare8 { ExternalWritable := 'False'} : DInt;
         dSpare9 { ExternalWritable := 'False'} : DInt;
         dSpare10 { ExternalWritable := 'False'} : DInt;
         dSpare11 { ExternalWritable := 'False'} : DInt;
         dSpare12 { ExternalWritable := 'False'} : DInt;
         dSpare13 { ExternalWritable := 'False'} : DInt;
         dSpare14 { ExternalWritable := 'False'} : DInt;
         dSpare15 { ExternalWritable := 'False'} : DInt;
         rSpare0 { ExternalWritable := 'False'} : Real;
         rSpare1 { ExternalWritable := 'False'} : Real;
         rSpare2 { ExternalWritable := 'False'} : Real;
         rSpare3 { ExternalWritable := 'False'} : Real;
         rSpare4 { ExternalWritable := 'False'} : Real;
         rSpare5 { ExternalWritable := 'False'} : Real;
         rSpare6 { ExternalWritable := 'False'} : Real;
         rSpare7 { ExternalWritable := 'False'} : Real;
         rSpare8 { ExternalWritable := 'False'} : Real;
         tManCmd { ExternalWritable := 'False'} : Struct
            xRunFdbk { ExternalWritable := 'False'} : Bool;   // Manual run fdbk {x|x|x|x|O}
            xSpare2 { ExternalWritable := 'False'} : Bool;
            xSpare3 { ExternalWritable := 'False'} : Bool;
            xSpare4 { ExternalWritable := 'False'} : Bool;
            xSpare5 { ExternalWritable := 'False'} : Bool;
            xSpare6 { ExternalWritable := 'False'} : Bool;
            xSpare7 { ExternalWritable := 'False'} : Bool;
            xSpare8 { ExternalWritable := 'False'} : Bool;
            xSpare9 { ExternalWritable := 'False'} : Bool;
            xSpare10 { ExternalWritable := 'False'} : Bool;
            xSpare11 { ExternalWritable := 'False'} : Bool;
            xSpare12 { ExternalWritable := 'False'} : Bool;
            xSpare13 { ExternalWritable := 'False'} : Bool;
            xSpare14 { ExternalWritable := 'False'} : Bool;
            xSpare15 { ExternalWritable := 'False'} : Bool;
            xSpare { ExternalWritable := 'False'} : Array[0..15] of Bool;
         END_STRUCT;
      END_STRUCT;
      tHMW : Struct   // HMI Write
         xEnableRunAlwaysModeBreaker : Bool;   // Enable run always breaker {x|x|x|x|O}
         xSpare1 : Bool;
         xSpare2 : Bool;
         xSpare3 : Bool;
         xSpare4 : Bool;
         xSpare5 : Bool;
         xSpare6 : Bool;
         xSpare7 : Bool;
         xSpare8 : Bool;
         xSpare9 : Bool;
         xSpare10 : Bool;   //
         xSpare11 : Bool;
         xSpare12 : Bool;
         xSpare13 : Bool;
         xEnableManualCommand : Bool;   // Enable Disable Manual command {x|x|x|x|O}
         xSpare15 : Bool;
         xSpare16 : Bool;
         xSpare17 : Bool;
         xSpare18 : Bool;
         xSpare19 : Bool;
         xSpare20 : Bool;
         xSpare21 : Bool;
         xSpare22 : Bool;
         xSpare23 : Bool;
         xSpare24 : Bool;
         xSpare25 : Bool;
         xSpare26 : Bool;
         xSpare27 : Bool;
         xSpare28 : Bool;
         xSpare29 : Bool;
         xSpare30 : Bool;
         xSpare31 : Bool;
         xSpare : Array[0..15] of Bool;
         iSpare0 : Int;
         iSpare1 : Int;
         iSpare2 : Int;
         iSpare3 : Int;
         iSpare4 : Int;
         iSpare5 : Int;
         iSpare6 : Int;
         iSpare7 : Int;
         iSpare8 : Int;
         iSpare9 : Int;
         iSpare10 : Int;
         iSpare11 : Int;
         iSpare12 : Int;
         iSpare13 : Int;
         iSpare14 : Int;
         iSpare15 : Int;
         iSpare16 : Int;
         dBreakerRetainTime_s : DInt;   // Breaker retain command after rise {ms|s|0|120|O}
         dSpare1 : DInt;
         dSpare2 : DInt;
         dSpare3 : DInt;
         dSpare4 : DInt;
         dSpare5 : DInt;
         dSpare6 : DInt;
         dSpare7 : DInt;
         dSpare8 : DInt;
         dSpare9 : DInt;
         dSpare10 : DInt;
         dSpare11 : DInt;
         dSpare12 : DInt;
         dSpare13 : DInt;
         dSpare14 : DInt;
         dSpare15 : DInt;
         dSpare16 : DInt;
         rSpare0 : Real;
         rSpare1 : Real;
         rSpare2 : Real;
         rSpare3 : Real;
         rSpare4 : Real;
         rSpare5 : Real;
         rSpare6 : Real;
         rSpare7 : Real;
         rSpare8 : Real;
         tManCmd : Struct
            xRun : Bool;   // Manual run {x|x|x|x|O}
            xSpare1 : Bool;
            xSpare2 { ExternalWritable := 'False'} : Bool;
            xSpare3 { ExternalWritable := 'False'} : Bool;
            xSpare4 { ExternalWritable := 'False'} : Bool;
            xSpare5 { ExternalWritable := 'False'} : Bool;
            xSpare6 { ExternalWritable := 'False'} : Bool;
            xSpare7 { ExternalWritable := 'False'} : Bool;
            xSpare8 { ExternalWritable := 'False'} : Bool;
            xSpare9 { ExternalWritable := 'False'} : Bool;
            xSpare10 { ExternalWritable := 'False'} : Bool;
            xSpare11 { ExternalWritable := 'False'} : Bool;
            xSpare12 { ExternalWritable := 'False'} : Bool;
            xSpare13 { ExternalWritable := 'False'} : Bool;
            xSpare14 { ExternalWritable := 'False'} : Bool;
            xSpare15 { ExternalWritable := 'False'} : Bool;
            xSpare16 : Bool;
            xSpare17 : Bool;
            xSpare18 : Bool;
            xSpare19 : Bool;
            xSpare20 : Bool;
            xSpare21 : Bool;
            xSpare22 : Bool;
            xSpare23 : Bool;
            xSpare24 : Bool;
            xSpare25 : Bool;
            xSpare26 : Bool;
            xSpare27 : Bool;
            xSpare28 : Bool;
            xSpare29 : Bool;
            xSpare30 : Bool;
            xSpare31 : Bool;
         END_STRUCT;
      END_STRUCT;
   END_STRUCT;


BEGIN
   tHMW.tManCmd.xRun := false;

END_DATA_BLOCK

DATA_BLOCK "DB_CrossCut_2_HMI"
{ DB_Accessible_From_OPC_UA := 'FALSE' ;
 DB_Accessible_From_Webserver := 'FALSE' ;
 S7_Optimized_Access := 'FALSE' }
VERSION : 0.1
NON_RETAIN
   STRUCT
      tALM : Struct   // HMI Alarms
         tE : Struct   // Emergency alarms
            xLocON : Bool;   // KE.Local emergency ON {X|X|X|X|O}
            xLocal1 : Bool;   // SB.Local emergency push button 1 {X|X|X|X|O}
            xLocal2 : Bool;   // SB.Local emergency push button 2 {X|X|X|X|O}
            xLocal3 : Bool;   // SB.Local emergency push button 3 {X|X|X|X|O}
            xSpare_4 : Bool;
            xSpare_5 : Bool;
            xSpare_6 : Bool;
            xSpare_7 : Bool;
            xSpare_8 : Bool;
            xSpare_9 : Bool;
            xSpare_10 : Bool;
            xSpare_11 : Bool;
            xSpare_12 : Bool;
            xSpare_13 : Bool;
            xSpare_14 : Bool;
            xSpare_15 : Bool;
            xSpare_16 : Bool;
            xSpare_17 : Bool;
            xSpare_18 : Bool;
            xSpare_19 : Bool;
            xSpare_20 : Bool;
            xSpare_21 : Bool;
            xSpare_22 : Bool;
            xSpare_23 : Bool;
            xSpare_24 : Bool;
            xSpare_25 : Bool;
            xSpare_26 : Bool;
            xSpare_27 : Bool;
            xSpare_28 : Bool;
            xSpare_29 : Bool;
            xSpare_30 : Bool;
            xSpare_31 : Bool;
         END_STRUCT;
         tS : Struct   // Stopping faults
            xAxisNotAvail : Bool;   // AZ.Axis not available {X|X|X|X|O}
            xInpInstallation : Bool;   // L+.Input power supply ON {X|X|X|X|O}
            xAuxPower : Bool;   // L+.Auxiliary power supple set-in {X|X|X|X|O}
            xAreaSafety : Bool;   // KE.Area safety {X|X|X|X|O}
            xOverstroke : Bool;   // KA.Carriage overstroke {X|X|X|X|O}
            xExternInputPower : Bool;   // L+.External input power supply {X|X|X|X|O}
            xCarriageCutOut : Bool;   // QM.Carriage translation overload {X|X|X|X|O}
            xDriveTrip : Bool;   // AZ.Drive trip {X|X|X|X|O}
            xDriveNotEnabled : Bool;   // AZ.Drive not enabled {X|X|X|X|O}
            xAxisNotReady : Bool;   // AZ.Axis not ready {X|X|X|X|O}
            xDriveNotReady : Bool;   // AZ.Drive not ready {X|X|X|X|O}
            xAxisNotSyncro : Bool;   // AZ.Axis not syncronized {X|X|X|X|O}
            xSpare_12 : Bool;
            xSpare_13 : Bool;
            xSpare_14 : Bool;
            xSpare_15 : Bool;
            xSpare_16 : Bool;
            xSpare_17 : Bool;
            xSpare_18 : Bool;
            xSpare_19 : Bool;
            xSpare_20 : Bool;
            xSpare_21 : Bool;
            xSpare_22 : Bool;
            xSpare_23 : Bool;
            xSpare_24 : Bool;
            xSpare_25 : Bool;
            xSpare_26 : Bool;
            xSpare_27 : Bool;
            xSpare_28 : Bool;
            xSpare_29 : Bool;
            xSpare_30 : Bool;
            xSpare_31 : Bool;
         END_STRUCT;
         tF : Struct   // Faults
            xSpare_0 : Bool;
            xSpare_1 : Bool;
            xSpare_2 : Bool;
            xSpare_3 : Bool;
            xSpare_4 : Bool;
            xSpare_5 : Bool;
            xSpare_6 : Bool;
            xSpare_7 : Bool;
            xSpare_8 : Bool;
            xSpare_9 : Bool;
            xSpare_10 : Bool;
            xSpare_11 : Bool;
            xSpare_12 : Bool;
            xSpare_13 : Bool;
            xSpare_14 : Bool;
            xSpare_15 : Bool;
            xSpare_16 : Bool;
            xSpare_17 : Bool;
            xSpare_18 : Bool;
            xSpare_19 : Bool;
            xSpare_20 : Bool;
            xSpare_21 : Bool;
            xSpare_22 : Bool;
            xSpare_23 : Bool;
            xSpare_24 : Bool;
            xSpare_25 : Bool;
            xSpare_26 : Bool;
            xSpare_27 : Bool;
            xSpare_28 : Bool;
            xSpare_29 : Bool;
            xSpare_30 : Bool;
            xSpare_31 : Bool;
         END_STRUCT;
         tW : Struct   // Warnings
            xSpare_0 : Bool;
            xSpare_1 : Bool;
            xSpare_2 : Bool;
            xSpare_3 : Bool;
            xSpare_4 : Bool;
            xSpare_5 : Bool;
            xSpare_6 : Bool;
            xSpare_7 : Bool;
            xSpare_8 : Bool;
            xSpare_9 : Bool;
            xSpare_10 : Bool;
            xSpare_11 : Bool;
            xSpare_12 : Bool;
            xSpare_13 : Bool;
            xSpare_14 : Bool;
            xSpare_15 : Bool;
            xSpare_16 : Bool;
            xSpare_17 : Bool;
            xSpare_18 : Bool;
            xSpare_19 : Bool;
            xSpare_20 : Bool;
            xSpare_21 : Bool;
            xSpare_22 : Bool;
            xSpare_23 : Bool;
            xSpare_24 : Bool;
            xSpare_25 : Bool;
            xSpare_26 : Bool;
            xSpare_27 : Bool;
            xSpare_28 : Bool;
            xSpare_29 : Bool;
            xSpare_30 : Bool;
            xSpare_31 : Bool;
         END_STRUCT;
      END_STRUCT;
      tHMR : Struct   // HMI Read
         xSpare0 : Bool;   //
         xSpare1 : Bool;   //
         xSpare2 : Bool;
         xSpare3 : Bool;
         xSpare4 : Bool;
         xSpare5 : Bool;
         xSpare6 : Bool;
         xSpare7 : Bool;
         xSpare8 : Bool;
         xSpare9 : Bool;
         xSpare10 : Bool;
         xSpare11 : Bool;
         xSpare12 : Bool;
         xSpare13 : Bool;
         xManualCommandEnabled : Bool;   // Manual Command enabled {x|x|x|x|O}
         xSpare15 : Bool;
         xSpare16 : Bool;
         xSpare17 : Bool;
         xSpare18 : Bool;
         xSpare19 : Bool;
         xSpare20 : Bool;
         xSpare21 : Bool;
         xSpare22 : Bool;
         xSpare23 : Bool;
         xSpare24 : Bool;
         xSpare25 : Bool;
         xSpare26 : Bool;
         xSpare27 : Bool;
         xSpare28 : Bool;
         xSpare29 : Bool;
         xSpare30 : Bool;
         xSpare31 : Bool;
         xSpare : Array[0..15] of Bool;
         iSpare0 { ExternalWritable := 'False'} : Int;
         iSpare1 { ExternalWritable := 'False'} : Int;
         iSpare2 { ExternalWritable := 'False'} : Int;
         iSpare3 { ExternalWritable := 'False'} : Int;
         iSpare4 { ExternalWritable := 'False'} : Int;
         iSpare5 { ExternalWritable := 'False'} : Int;
         iSpare6 { ExternalWritable := 'False'} : Int;
         iSpare7 { ExternalWritable := 'False'} : Int;
         iSpare8 { ExternalWritable := 'False'} : Int;
         iSpare9 { ExternalWritable := 'False'} : Int;
         iSpare10 { ExternalWritable := 'False'} : Int;
         iSpare11 { ExternalWritable := 'False'} : Int;
         iSpare12 { ExternalWritable := 'False'} : Int;
         iSpare13 { ExternalWritable := 'False'} : Int;
         iSpare14 { ExternalWritable := 'False'} : Int;
         iSpare15 { ExternalWritable := 'False'} : Int;
         iSpare16 { ExternalWritable := 'False'} : Int;
         dDistanceSnaproll_cmm { ExternalWritable := 'False'} : DInt;   // Distance from snaproll [mm/100] {mm/100|mm|x|x|M}
         dStatus { ExternalWritable := 'False'} : DInt;   // XCut actual status (1=Idle 3=Running 7=Faulted)  {X|X|X|X|O}
         dXCutActualStatus { ExternalWritable := 'False'} : DInt;   // XCut actual status (1=Disabled 3=Enabled) {X|X|X|X|O}
         dXCutStatusRequest { ExternalWritable := 'False'} : DInt;   // XCut status request (1=Disabled 3=Enabled) {X|X|X|X|O}
         dDistanceFromCenterLine_cmm { ExternalWritable := 'False'} : DInt;   // Distance from center line [mm/100] {mm/100|mm|X|X|O}
         dAngleValue_uDegree { ExternalWritable := 'False'} : DInt;   // Angle value [°/1000000] {°/1000000|°|X|X|O}
         dActualCutPosRequest { ExternalWritable := 'False'} : DInt;   // Actual cut position request (1=By operator 2=On gross ribbon 3=On net ribbon 4=On YCut position) {X|X|X|X|O}
         dCarriagePosition_cmm { ExternalWritable := 'False'} : DInt;   // Actual carriage position [mm/100]
         dSpare8 { ExternalWritable := 'False'} : DInt;
         dSpare9 { ExternalWritable := 'False'} : DInt;
         dSpare10 { ExternalWritable := 'False'} : DInt;
         dSpare11 { ExternalWritable := 'False'} : DInt;
         dSpare12 { ExternalWritable := 'False'} : DInt;
         dSpare13 { ExternalWritable := 'False'} : DInt;
         dSpare14 { ExternalWritable := 'False'} : DInt;
         dSpare15 { ExternalWritable := 'False'} : DInt;
         rHeadUsage_km { ExternalWritable := 'False'} : Real;   // Head usage [Km] {Km|Km|X|X|O}
         rSpare1 { ExternalWritable := 'False'} : Real;
         rSpare2 { ExternalWritable := 'False'} : Real;
         rSpare3 { ExternalWritable := 'False'} : Real;
         rSpare4 { ExternalWritable := 'False'} : Real;
         rSpare5 { ExternalWritable := 'False'} : Real;
         rSpare6 { ExternalWritable := 'False'} : Real;
         rSpare7 { ExternalWritable := 'False'} : Real;
         rSpare8 { ExternalWritable := 'False'} : Real;
         tManCmd { ExternalWritable := 'False'} : Struct
            xManJogFwdFdbk { ExternalWritable := 'False'} : Bool;   // Manual jog forward feedback {X|X|X|X|O}
            xManJogBckFdbk { ExternalWritable := 'False'} : Bool;   // Manual jog backward feedback {X|X|X|X|O}
            xManCarriageDownFdbk { ExternalWritable := 'False'} : Bool;   // Manual carriage down feedback {X|X|X|X|O}
            xManFireONFdbk { ExternalWritable := 'False'} : Bool;   // Manual fire ON feedback {X|X|X|X|O}
            xManOilONFdbk { ExternalWritable := 'False'} : Bool;   // Manual oil ON feedback {X|X|X|X|O}
            xSpare5 { ExternalWritable := 'False'} : Bool;
            xSpare6 { ExternalWritable := 'False'} : Bool;
            xSpare7 { ExternalWritable := 'False'} : Bool;
            xSpare8 { ExternalWritable := 'False'} : Bool;
            xSpare9 { ExternalWritable := 'False'} : Bool;
            xSpare10 { ExternalWritable := 'False'} : Bool;
            xSpare11 { ExternalWritable := 'False'} : Bool;
            xSpare12 { ExternalWritable := 'False'} : Bool;
            xSpare13 { ExternalWritable := 'False'} : Bool;
            xSpare14 { ExternalWritable := 'False'} : Bool;
            xSpare15 { ExternalWritable := 'False'} : Bool;
            xSpare { ExternalWritable := 'False'} : Array[0..15] of Bool;
         END_STRUCT;
      END_STRUCT;
      tHMW : Struct   // HMI Write
         xCutBreakEnabled { ExternalWritable := 'False'} : Bool;   // Cut on glass break enabled {X|X|X|X|O}
         xIncAngleValue : Bool;   // Increment angle value {X|X|X|X|O}
         xDecAngleValue : Bool;   // Decrement angle value {X|X|X|X|O}
         xCalibDistRequest : Bool;   // Calibration distance request {X|X|X|X|O}
         xCalibDiagRequest : Bool;   // Calibration diagonal request {X|X|X|X|O}
         xCutOperator : Bool;   // Cutting position by operator request {X|X|X|X|O}
         xCutGross : Bool;   // Cutting position by gross width position {X|X|X|X|O}
         xCutNet : Bool;   // Cutting position by net width position {X|X|X|X|O}
         xCutYCut : Bool;   // Cutting position by YCut position {X|X|X|X|O}
         xSpare9 : Bool;
         xSpare10 : Bool;
         xSpare11 : Bool;
         xSpare12 : Bool;
         xResetHeadUsage : Bool;   // Reset the head usage {X|X|X|X|O}
         xEnableManualCommand : Bool;   // Enable Disable Manual command {x|x|x|x|O}
         xUpdateDistanceSnaproll : Bool;   // Update distance from snaproll {x|x|x|x|M}
         xUpdateDistCenterLine : Bool;   // Update distance from center line {X|X|X|X|M}
         xUpdateAngleValue : Bool;   // Update angle value {X|X|X|X|M}
         xSpare18 : Bool;
         xSpare19 : Bool;
         xSpare20 : Bool;
         xSpare21 : Bool;
         xSpare22 : Bool;
         xSpare23 : Bool;
         xSpare24 : Bool;
         xSpare25 : Bool;
         xSpare26 : Bool;
         xSpare27 : Bool;
         xSpare28 : Bool;
         xSpare29 : Bool;
         xSpare30 : Bool;
         xSpare31 : Bool;
         xSpare : Array[0..15] of Bool;
         iSpare0 : Int;
         iSpare1 : Int;
         iSpare2 : Int;
         iSpare3 : Int;
         iSpare4 : Int;
         iSpare5 : Int;
         iSpare6 : Int;
         iSpare7 : Int;
         iSpare8 : Int;
         iSpare9 : Int;
         iSpare10 : Int;
         iSpare11 : Int;
         iSpare12 : Int;
         iSpare13 : Int;
         iSpare14 : Int;
         iSpare15 : Int;
         iSpare16 : Int;
         dDistanceSnaproll_cmm : DInt;   // Distance from snaproll [mm/100] {mm/100|mm|1|70000|M}
         dDistanceFromCenterLine_cmm : DInt;   // Distance from center line [mm/100] {mm/100|mm|-3000|0|M}
         dAngleValue_uDegree : DInt;   // Bridge angle value [°/1000000] {°/1000000|°|7|9|M}
         dOperStartCutPos_cmm : DInt;   // Operator start cut position [mm/100] {mm/100|mm|-3000|0|O}
         dOperEndCutPos_cmm : DInt;   // Operator end cut position  [mm/100] {mm/100|mm|0|3000|O}
         dDescReactTime_ms : DInt;   // Carriage descent reaction time [ms] {ms|s|0|1|M}
         dRaiseReactTime_ms : DInt;   // Carriage raise reaction time [ms] {ms|s|0|1|M}
         dFireONReactTime_ms : DInt;   // Fire ON reaction time [ms] {ms|s|0|1|M}
         dFireOFFReactTime_ms : DInt;   // Fire OFF reaction time [ms] {ms|s|0|1|M}
         dOilONDelay_ms : DInt;   // Oil ON delay [ms] {ms|s|-1|1|O}
         dOilOFFDelay_ms : DInt;   // Oil OFF delay [ms] {ms|s|-1|1|O}
         dCutStartOffsetDelay_cmm : DInt;   // Start cut offset delay [mm/100] {mm/100|mm|-500|500|O}
         dCutEndOffsetDelay_cmm : DInt;   // End cut offset delay [mm/100] {mm/100|mm|-500|500|O}
         dDistTeoLength_cmm : DInt;   // Calibration distance.Theorical length [mm/100] {mm/100|mm|0|7000|O}
         dDistRealLength_cmm : DInt;   // Calibration distance.Real length [mm/100] {mm/100|mm|0|7000|O}
         dDiagRealLength_cmm : DInt;   // Calibration diagonal.Real length [mm/100] {mm/100|mm|0|7000|O}
         dDiagRealWidth_cmm : DInt;   // Calibration diagonal.Real width [mm/100] {mm/100|mm|0|4000|O}
         dDiagGlassFlow_cmm : DInt;   // Calibration diagonal.Real length diagonal glass flow [mm/100] {mm/100|mm|0|10000|O}
         dDiagGlassOppFlow_cmm : DInt;   // Calibration diagonal.Real length diagonal opposite glass flow [mm/100] {mm/100|mm|0|10000|O}
         dCuttingPressure_mN : DInt;   // Cutting pressure [N/1000] {N/1000|N|9|180|O}
         dPosOffset_cmm : DInt;   // Calibration offset distance from snaproll [mm/100]  {mm/100|mm|-50|50|O}
         dCutPriority : DInt;   // Cut priority number  {X|X|0|5|O}
         dSpare22 : DInt;
         rSpare6 : Real;
         rSpare7 : Real;
         rSpare8 : Real;
         tManCmd : Struct
            xMan_JogForward : Bool;   // Manual mode - Jog forward {X|X|X|X|M}
            xMan_JobBackward : Bool;   // Manual mode - Jog backward {X|X|X|X|M}
            xMan_CarriageDown : Bool;   // Manual mode - Carriage down {X|X|X|X|M}
            xMan_FireOn : Bool;   // Manual mode - Fire ON {X|X|X|X|M}
            xMan_OilOn : Bool;   // Manual mode - Oil ON {X|X|X|X|M}
            xSpare5 { ExternalWritable := 'False'} : Bool;
            xSpare6 { ExternalWritable := 'False'} : Bool;
            xSpare7 { ExternalWritable := 'False'} : Bool;
            xSpare8 { ExternalWritable := 'False'} : Bool;
            xSpare9 { ExternalWritable := 'False'} : Bool;
            xSpare10 { ExternalWritable := 'False'} : Bool;
            xSpare11 { ExternalWritable := 'False'} : Bool;
            xSpare12 { ExternalWritable := 'False'} : Bool;
            xSpare13 { ExternalWritable := 'False'} : Bool;
            xSpare14 { ExternalWritable := 'False'} : Bool;
            xSpare15 { ExternalWritable := 'False'} : Bool;
            xSpare16 : Bool;
            xSpare17 : Bool;
            xSpare18 : Bool;
            xSpare19 : Bool;
            xSpare20 : Bool;
            xSpare21 : Bool;
            xSpare22 : Bool;
            xSpare23 : Bool;
            xSpare24 : Bool;
            xSpare25 : Bool;
            xSpare26 : Bool;
            xSpare27 : Bool;
            xSpare28 : Bool;
            xSpare29 : Bool;
            xSpare30 : Bool;
            xSpare31 : Bool;
         END_STRUCT;
      END_STRUCT;
   END_STRUCT;


BEGIN

END_DATA_BLOCK

DATA_BLOCK "DB_Marker_HMI"
{ DB_Accessible_From_OPC_UA := 'FALSE' ;
 DB_Accessible_From_Webserver := 'FALSE' ;
 S7_Optimized_Access := 'FALSE' }
VERSION : 0.1
NON_RETAIN
   STRUCT
      tALM { ExternalWritable := 'False'} : Struct   // HMI Alarms
         tE { ExternalWritable := 'False'} : Struct   // Stopping faults
            xSpare_0 { ExternalWritable := 'False'} : Bool;
            xSpare_1 { ExternalWritable := 'False'} : Bool;
            xSpare_2 { ExternalWritable := 'False'} : Bool;
            xSpare_3 { ExternalWritable := 'False'} : Bool;
            xSpare_4 { ExternalWritable := 'False'} : Bool;
            xSpare_5 { ExternalWritable := 'False'} : Bool;
            xSpare_6 { ExternalWritable := 'False'} : Bool;
            xSpare_7 { ExternalWritable := 'False'} : Bool;
            xSpare_8 { ExternalWritable := 'False'} : Bool;
            xSpare_9 { ExternalWritable := 'False'} : Bool;
            xSpare_10 { ExternalWritable := 'False'} : Bool;
            xSpare_11 { ExternalWritable := 'False'} : Bool;
            xSpare_12 { ExternalWritable := 'False'} : Bool;
            xSpare_13 { ExternalWritable := 'False'} : Bool;
            xSpare_14 { ExternalWritable := 'False'} : Bool;
            xSpare_15 { ExternalWritable := 'False'} : Bool;
            xSpare_16 { ExternalWritable := 'False'} : Bool;
            xSpare_17 { ExternalWritable := 'False'} : Bool;
            xSpare_18 { ExternalWritable := 'False'} : Bool;
            xSpare_19 { ExternalWritable := 'False'} : Bool;
            xSpare_20 { ExternalWritable := 'False'} : Bool;
            xSpare_21 { ExternalWritable := 'False'} : Bool;
            xSpare_22 { ExternalWritable := 'False'} : Bool;
            xSpare_23 { ExternalWritable := 'False'} : Bool;
            xSpare_24 { ExternalWritable := 'False'} : Bool;
            xSpare_25 { ExternalWritable := 'False'} : Bool;
            xSpare_26 { ExternalWritable := 'False'} : Bool;
            xSpare_27 { ExternalWritable := 'False'} : Bool;
            xSpare_28 { ExternalWritable := 'False'} : Bool;
            xSpare_29 { ExternalWritable := 'False'} : Bool;
            xSpare_30 { ExternalWritable := 'False'} : Bool;
            xSpare_31 { ExternalWritable := 'False'} : Bool;
         END_STRUCT;
         tS { ExternalWritable := 'False'} : Struct   // Stopping faults
            xTOutSendData { ExternalWritable := 'False'} : Bool;   // Timeout send data to bridge
            xSpare_1 { ExternalAccessible := 'False'; ExternalVisible := 'False'; ExternalWritable := 'False'} : Bool;
            xSpare_2 { ExternalAccessible := 'False'; ExternalVisible := 'False'; ExternalWritable := 'False'} : Bool;
            xSpare_3 { ExternalAccessible := 'False'; ExternalVisible := 'False'; ExternalWritable := 'False'} : Bool;
            xSpare_4 { ExternalAccessible := 'False'; ExternalVisible := 'False'; ExternalWritable := 'False'} : Bool;
            xSpare_5 { ExternalAccessible := 'False'; ExternalVisible := 'False'; ExternalWritable := 'False'} : Bool;
            xSpare_6 { ExternalAccessible := 'False'; ExternalVisible := 'False'; ExternalWritable := 'False'} : Bool;
            xSpare_7 { ExternalAccessible := 'False'; ExternalVisible := 'False'; ExternalWritable := 'False'} : Bool;
            xSpare_8 { ExternalAccessible := 'False'; ExternalVisible := 'False'; ExternalWritable := 'False'} : Bool;
            xSpare_9 { ExternalAccessible := 'False'; ExternalVisible := 'False'; ExternalWritable := 'False'} : Bool;
            xSpare_10 { ExternalAccessible := 'False'; ExternalVisible := 'False'; ExternalWritable := 'False'} : Bool;
            xSpare_11 { ExternalAccessible := 'False'; ExternalVisible := 'False'; ExternalWritable := 'False'} : Bool;
            xSpare_12 { ExternalAccessible := 'False'; ExternalVisible := 'False'; ExternalWritable := 'False'} : Bool;
            xSpare_13 { ExternalAccessible := 'False'; ExternalVisible := 'False'; ExternalWritable := 'False'} : Bool;
            xSpare_14 { ExternalAccessible := 'False'; ExternalVisible := 'False'; ExternalWritable := 'False'} : Bool;
            xSpare_15 { ExternalAccessible := 'False'; ExternalVisible := 'False'; ExternalWritable := 'False'} : Bool;
            xSpare_16 { ExternalAccessible := 'False'; ExternalVisible := 'False'; ExternalWritable := 'False'} : Bool;
            xSpare_17 { ExternalAccessible := 'False'; ExternalVisible := 'False'; ExternalWritable := 'False'} : Bool;
            xSpare_18 { ExternalAccessible := 'False'; ExternalVisible := 'False'; ExternalWritable := 'False'} : Bool;
            xSpare_19 { ExternalAccessible := 'False'; ExternalVisible := 'False'; ExternalWritable := 'False'} : Bool;
            xSpare_20 { ExternalAccessible := 'False'; ExternalVisible := 'False'; ExternalWritable := 'False'} : Bool;
            xSpare_21 { ExternalAccessible := 'False'; ExternalVisible := 'False'; ExternalWritable := 'False'} : Bool;
            xSpare_22 { ExternalAccessible := 'False'; ExternalVisible := 'False'; ExternalWritable := 'False'} : Bool;
            xSpare_23 { ExternalAccessible := 'False'; ExternalVisible := 'False'; ExternalWritable := 'False'} : Bool;
            xSpare_24 { ExternalAccessible := 'False'; ExternalVisible := 'False'; ExternalWritable := 'False'} : Bool;
            xSpare_25 { ExternalAccessible := 'False'; ExternalVisible := 'False'; ExternalWritable := 'False'} : Bool;
            xSpare_26 { ExternalAccessible := 'False'; ExternalVisible := 'False'; ExternalWritable := 'False'} : Bool;
            xSpare_27 { ExternalAccessible := 'False'; ExternalVisible := 'False'; ExternalWritable := 'False'} : Bool;
            xSpare_28 { ExternalAccessible := 'False'; ExternalVisible := 'False'; ExternalWritable := 'False'} : Bool;
            xSpare_29 { ExternalAccessible := 'False'; ExternalVisible := 'False'; ExternalWritable := 'False'} : Bool;
            xSpare_30 { ExternalAccessible := 'False'; ExternalVisible := 'False'; ExternalWritable := 'False'} : Bool;
            xSpare_31 { ExternalAccessible := 'False'; ExternalVisible := 'False'; ExternalWritable := 'False'} : Bool;
         END_STRUCT;
         tF { ExternalAccessible := 'False'; ExternalVisible := 'False'; ExternalWritable := 'False'} : Struct   // Faults
            xSpare_0 { ExternalAccessible := 'False'; ExternalVisible := 'False'; ExternalWritable := 'False'} : Bool;
            xSpare_1 { ExternalAccessible := 'False'; ExternalVisible := 'False'; ExternalWritable := 'False'} : Bool;
            xSpare_2 { ExternalAccessible := 'False'; ExternalVisible := 'False'; ExternalWritable := 'False'} : Bool;
            xSpare_3 { ExternalAccessible := 'False'; ExternalVisible := 'False'; ExternalWritable := 'False'} : Bool;
            xSpare_4 { ExternalAccessible := 'False'; ExternalVisible := 'False'; ExternalWritable := 'False'} : Bool;
            xSpare_5 { ExternalAccessible := 'False'; ExternalVisible := 'False'; ExternalWritable := 'False'} : Bool;
            xSpare_6 { ExternalAccessible := 'False'; ExternalVisible := 'False'; ExternalWritable := 'False'} : Bool;
            xSpare_7 { ExternalAccessible := 'False'; ExternalVisible := 'False'; ExternalWritable := 'False'} : Bool;
            xSpare_8 { ExternalAccessible := 'False'; ExternalVisible := 'False'; ExternalWritable := 'False'} : Bool;
            xSpare_9 { ExternalAccessible := 'False'; ExternalVisible := 'False'; ExternalWritable := 'False'} : Bool;
            xSpare_10 { ExternalAccessible := 'False'; ExternalVisible := 'False'; ExternalWritable := 'False'} : Bool;
            xSpare_11 { ExternalAccessible := 'False'; ExternalVisible := 'False'; ExternalWritable := 'False'} : Bool;
            xSpare_12 { ExternalAccessible := 'False'; ExternalVisible := 'False'; ExternalWritable := 'False'} : Bool;
            xSpare_13 { ExternalAccessible := 'False'; ExternalVisible := 'False'; ExternalWritable := 'False'} : Bool;
            xSpare_14 { ExternalAccessible := 'False'; ExternalVisible := 'False'; ExternalWritable := 'False'} : Bool;
            xSpare_15 { ExternalAccessible := 'False'; ExternalVisible := 'False'; ExternalWritable := 'False'} : Bool;
            xSpare_16 { ExternalAccessible := 'False'; ExternalVisible := 'False'; ExternalWritable := 'False'} : Bool;
            xSpare_17 { ExternalAccessible := 'False'; ExternalVisible := 'False'; ExternalWritable := 'False'} : Bool;
            xSpare_18 { ExternalAccessible := 'False'; ExternalVisible := 'False'; ExternalWritable := 'False'} : Bool;
            xSpare_19 { ExternalAccessible := 'False'; ExternalVisible := 'False'; ExternalWritable := 'False'} : Bool;
            xSpare_20 { ExternalAccessible := 'False'; ExternalVisible := 'False'; ExternalWritable := 'False'} : Bool;
            xSpare_21 { ExternalAccessible := 'False'; ExternalVisible := 'False'; ExternalWritable := 'False'} : Bool;
            xSpare_22 { ExternalAccessible := 'False'; ExternalVisible := 'False'; ExternalWritable := 'False'} : Bool;
            xSpare_23 { ExternalAccessible := 'False'; ExternalVisible := 'False'; ExternalWritable := 'False'} : Bool;
            xSpare_24 { ExternalAccessible := 'False'; ExternalVisible := 'False'; ExternalWritable := 'False'} : Bool;
            xSpare_25 { ExternalAccessible := 'False'; ExternalVisible := 'False'; ExternalWritable := 'False'} : Bool;
            xSpare_26 { ExternalAccessible := 'False'; ExternalVisible := 'False'; ExternalWritable := 'False'} : Bool;
            xSpare_27 { ExternalAccessible := 'False'; ExternalVisible := 'False'; ExternalWritable := 'False'} : Bool;
            xSpare_28 { ExternalAccessible := 'False'; ExternalVisible := 'False'; ExternalWritable := 'False'} : Bool;
            xSpare_29 { ExternalAccessible := 'False'; ExternalVisible := 'False'; ExternalWritable := 'False'} : Bool;
            xSpare_30 { ExternalAccessible := 'False'; ExternalVisible := 'False'; ExternalWritable := 'False'} : Bool;
            xSpare_31 { ExternalAccessible := 'False'; ExternalVisible := 'False'; ExternalWritable := 'False'} : Bool;
         END_STRUCT;
         tW { ExternalAccessible := 'False'; ExternalVisible := 'False'; ExternalWritable := 'False'} : Struct   // Warnings
            xSpare_0 { ExternalAccessible := 'False'; ExternalVisible := 'False'; ExternalWritable := 'False'} : Bool;
            xSpare_1 { ExternalAccessible := 'False'; ExternalVisible := 'False'; ExternalWritable := 'False'} : Bool;
            xSpare_2 { ExternalAccessible := 'False'; ExternalVisible := 'False'; ExternalWritable := 'False'} : Bool;
            xSpare_3 { ExternalAccessible := 'False'; ExternalVisible := 'False'; ExternalWritable := 'False'} : Bool;
            xSpare_4 { ExternalAccessible := 'False'; ExternalVisible := 'False'; ExternalWritable := 'False'} : Bool;
            xSpare_5 { ExternalAccessible := 'False'; ExternalVisible := 'False'; ExternalWritable := 'False'} : Bool;
            xSpare_6 { ExternalAccessible := 'False'; ExternalVisible := 'False'; ExternalWritable := 'False'} : Bool;
            xSpare_7 { ExternalAccessible := 'False'; ExternalVisible := 'False'; ExternalWritable := 'False'} : Bool;
            xSpare_8 { ExternalAccessible := 'False'; ExternalVisible := 'False'; ExternalWritable := 'False'} : Bool;
            xSpare_9 { ExternalAccessible := 'False'; ExternalVisible := 'False'; ExternalWritable := 'False'} : Bool;
            xSpare_10 { ExternalAccessible := 'False'; ExternalVisible := 'False'; ExternalWritable := 'False'} : Bool;
            xSpare_11 { ExternalAccessible := 'False'; ExternalVisible := 'False'; ExternalWritable := 'False'} : Bool;
            xSpare_12 { ExternalAccessible := 'False'; ExternalVisible := 'False'; ExternalWritable := 'False'} : Bool;
            xSpare_13 { ExternalAccessible := 'False'; ExternalVisible := 'False'; ExternalWritable := 'False'} : Bool;
            xSpare_14 { ExternalAccessible := 'False'; ExternalVisible := 'False'; ExternalWritable := 'False'} : Bool;
            xSpare_15 { ExternalAccessible := 'False'; ExternalVisible := 'False'; ExternalWritable := 'False'} : Bool;
            xSpare_16 { ExternalAccessible := 'False'; ExternalVisible := 'False'; ExternalWritable := 'False'} : Bool;
            xSpare_17 { ExternalAccessible := 'False'; ExternalVisible := 'False'; ExternalWritable := 'False'} : Bool;
            xSpare_18 { ExternalAccessible := 'False'; ExternalVisible := 'False'; ExternalWritable := 'False'} : Bool;
            xSpare_19 { ExternalAccessible := 'False'; ExternalVisible := 'False'; ExternalWritable := 'False'} : Bool;
            xSpare_20 { ExternalAccessible := 'False'; ExternalVisible := 'False'; ExternalWritable := 'False'} : Bool;
            xSpare_21 { ExternalAccessible := 'False'; ExternalVisible := 'False'; ExternalWritable := 'False'} : Bool;
            xSpare_22 { ExternalAccessible := 'False'; ExternalVisible := 'False'; ExternalWritable := 'False'} : Bool;
            xSpare_23 { ExternalAccessible := 'False'; ExternalVisible := 'False'; ExternalWritable := 'False'} : Bool;
            xSpare_24 { ExternalAccessible := 'False'; ExternalVisible := 'False'; ExternalWritable := 'False'} : Bool;
            xSpare_25 { ExternalAccessible := 'False'; ExternalVisible := 'False'; ExternalWritable := 'False'} : Bool;
            xSpare_26 { ExternalAccessible := 'False'; ExternalVisible := 'False'; ExternalWritable := 'False'} : Bool;
            xSpare_27 { ExternalAccessible := 'False'; ExternalVisible := 'False'; ExternalWritable := 'False'} : Bool;
            xSpare_28 { ExternalAccessible := 'False'; ExternalVisible := 'False'; ExternalWritable := 'False'} : Bool;
            xSpare_29 { ExternalAccessible := 'False'; ExternalVisible := 'False'; ExternalWritable := 'False'} : Bool;
            xSpare_30 { ExternalAccessible := 'False'; ExternalVisible := 'False'; ExternalWritable := 'False'} : Bool;
            xSpare_31 { ExternalAccessible := 'False'; ExternalVisible := 'False'; ExternalWritable := 'False'} : Bool;
         END_STRUCT;
      END_STRUCT;
      tHMR { ExternalWritable := 'False'} : Struct   // HMI Read
         xSpare0 { ExternalWritable := 'False'} : Bool;
         xSpare1 { ExternalWritable := 'False'} : Bool;
         xSpare2 { ExternalWritable := 'False'} : Bool;
         xSpare3 { ExternalWritable := 'False'} : Bool;
         xSpare4 { ExternalWritable := 'False'} : Bool;
         xSpare5 { ExternalWritable := 'False'} : Bool;
         xSpare6 { ExternalWritable := 'False'} : Bool;
         xSpare7 { ExternalWritable := 'False'} : Bool;
         xSpare8 { ExternalWritable := 'False'} : Bool;
         xSpare9 { ExternalWritable := 'False'} : Bool;
         xSpare10 { ExternalWritable := 'False'} : Bool;
         xSpare11 { ExternalWritable := 'False'} : Bool;
         xSpare12 { ExternalWritable := 'False'} : Bool;
         xSpare13 { ExternalWritable := 'False'} : Bool;
         xSpare14 { ExternalWritable := 'False'} : Bool;   //
         xSpare15 { ExternalWritable := 'False'} : Bool;
         xSpare16 { ExternalWritable := 'False'} : Bool;
         xSpare17 { ExternalWritable := 'False'} : Bool;
         xSpare18 { ExternalWritable := 'False'} : Bool;
         xSpare19 { ExternalWritable := 'False'} : Bool;
         xSpare20 { ExternalWritable := 'False'} : Bool;
         xSpare21 { ExternalWritable := 'False'} : Bool;
         xSpare22 { ExternalWritable := 'False'} : Bool;
         xSpare23 { ExternalWritable := 'False'} : Bool;
         xSpare24 { ExternalWritable := 'False'} : Bool;
         xSpare25 { ExternalWritable := 'False'} : Bool;
         xSpare26 { ExternalWritable := 'False'} : Bool;
         xSpare27 { ExternalWritable := 'False'} : Bool;
         xSpare28 { ExternalWritable := 'False'} : Bool;
         xSpare29 { ExternalWritable := 'False'} : Bool;
         xSpare30 { ExternalWritable := 'False'} : Bool;
         xSpare31 { ExternalWritable := 'False'} : Bool;
         xSpare { ExternalWritable := 'False'} : Array[0..15] of Bool;
         iSpare0 { ExternalWritable := 'False'} : Int;
         iSpare1 { ExternalWritable := 'False'} : Int;
         iSpare2 { ExternalWritable := 'False'} : Int;
         iSpare3 { ExternalWritable := 'False'} : Int;
         iSpare4 { ExternalWritable := 'False'} : Int;
         iSpare5 { ExternalWritable := 'False'} : Int;
         iSpare6 { ExternalWritable := 'False'} : Int;
         iSpare7 { ExternalWritable := 'False'} : Int;
         iSpare8 { ExternalWritable := 'False'} : Int;
         iSpare9 { ExternalWritable := 'False'} : Int;
         iSpare10 { ExternalWritable := 'False'} : Int;
         iSpare11 { ExternalWritable := 'False'} : Int;
         iSpare12 { ExternalWritable := 'False'} : Int;
         iSpare13 { ExternalWritable := 'False'} : Int;
         iSpare14 { ExternalWritable := 'False'} : Int;
         iSpare15 { ExternalWritable := 'False'} : Int;
         iSpare16 { ExternalWritable := 'False'} : Int;
         dSpare0 { ExternalWritable := 'False'} : DInt;
         dSpare1 { ExternalWritable := 'False'} : DInt;
         dSpare2 { ExternalWritable := 'False'} : DInt;
         dSpare3 { ExternalWritable := 'False'} : DInt;
         dSpare4 { ExternalWritable := 'False'} : DInt;
         dSpare5 { ExternalWritable := 'False'} : DInt;
         dSpare6 { ExternalWritable := 'False'} : DInt;
         dSpare7 { ExternalWritable := 'False'} : DInt;
         dSpare8 { ExternalWritable := 'False'} : DInt;
         dSpare9 { ExternalWritable := 'False'} : DInt;
         dSpare10 { ExternalWritable := 'False'} : DInt;
         dSpare11 { ExternalWritable := 'False'} : DInt;
         dSpare12 { ExternalWritable := 'False'} : DInt;
         dSpare13 { ExternalWritable := 'False'} : DInt;
         dSpare14 { ExternalWritable := 'False'} : DInt;
         dSpare15 { ExternalWritable := 'False'} : DInt;
         rSpare0 { ExternalWritable := 'False'} : Real;
         rSpare1 { ExternalWritable := 'False'} : Real;
         rSpare2 { ExternalWritable := 'False'} : Real;
         rSpare3 { ExternalWritable := 'False'} : Real;
         rSpare4 { ExternalWritable := 'False'} : Real;
         rSpare5 { ExternalWritable := 'False'} : Real;
         rSpare6 { ExternalWritable := 'False'} : Real;
         rSpare7 { ExternalWritable := 'False'} : Real;
         rSpare8 { ExternalWritable := 'False'} : Real;
         tManCmd { ExternalWritable := 'False'} : Struct
            xSpare0 { ExternalWritable := 'False'} : Bool;
            xSpare1 { ExternalWritable := 'False'} : Bool;
            xSpare2 { ExternalWritable := 'False'} : Bool;
            xSpare3 { ExternalWritable := 'False'} : Bool;
            xSpare4 { ExternalWritable := 'False'} : Bool;
            xSpare5 { ExternalWritable := 'False'} : Bool;
            xSpare6 { ExternalWritable := 'False'} : Bool;
            xSpare7 { ExternalWritable := 'False'} : Bool;
            xSpare8 { ExternalWritable := 'False'} : Bool;
            xSpare9 { ExternalWritable := 'False'} : Bool;
            xSpare10 { ExternalWritable := 'False'} : Bool;
            xSpare11 { ExternalWritable := 'False'} : Bool;
            xSpare12 { ExternalWritable := 'False'} : Bool;
            xSpare13 { ExternalWritable := 'False'} : Bool;
            xSpare14 { ExternalWritable := 'False'} : Bool;
            xSpare15 { ExternalWritable := 'False'} : Bool;
            xSpare { ExternalWritable := 'False'} : Array[0..15] of Bool;
         END_STRUCT;
      END_STRUCT;
      tHMW : Struct   // HMI Write
         xSpare0 : Bool;   //
         xSpare1 : Bool;
         xSpare2 : Bool;
         xSpare3 : Bool;
         xSpare4 : Bool;
         xSpare5 : Bool;
         xSpare6 : Bool;
         xSpare7 : Bool;
         xSpare8 : Bool;
         xSpare9 : Bool;
         xSpare10 : Bool;   //
         xSpare11 : Bool;
         xSpare12 : Bool;
         xSpare13 : Bool;
         xSpare14 : Bool;   //
         xSpare15 : Bool;
         xSpare16 : Bool;
         xSpare17 : Bool;
         xSpare18 : Bool;
         xSpare19 : Bool;
         xSpare20 : Bool;
         xSpare21 : Bool;
         xSpare22 : Bool;
         xSpare23 : Bool;
         xSpare24 : Bool;
         xSpare25 : Bool;
         xSpare26 : Bool;
         xSpare27 : Bool;
         xSpare28 : Bool;
         xSpare29 : Bool;
         xSpare30 : Bool;
         xSpare31 : Bool;
         xSpare : Array[0..15] of Bool;
         iSpare0 : Int;
         iSpare1 : Int;
         iSpare2 : Int;
         iSpare3 : Int;
         iSpare4 : Int;
         iSpare5 : Int;
         iSpare6 : Int;
         iSpare7 : Int;
         iSpare8 : Int;
         iSpare9 : Int;
         iSpare10 : Int;
         iSpare11 : Int;
         iSpare12 : Int;
         iSpare13 : Int;
         iSpare14 : Int;
         iSpare15 : Int;
         iSpare16 : Int;
         dSpare0 : DInt;   //
         dSpare1 : DInt;   //
         dSpare2 : DInt;   //
         dSpare3 : DInt;
         dSpare4 : DInt;
         dSpare5 : DInt;
         dSpare6 : DInt;
         dSpare7 : DInt;
         dSpare8 : DInt;
         dSpare9 : DInt;
         dSpare10 : DInt;
         dSpare11 : DInt;
         dSpare12 : DInt;
         dSpare13 : DInt;
         dSpare14 : DInt;
         dSpare15 : DInt;
         dSpare16 : DInt;
         rSpare0 : Real;
         rSpare1 : Real;
         rSpare2 : Real;
         rSpare3 : Real;
         rSpare4 : Real;
         rSpare5 : Real;
         rSpare6 : Real;
         rSpare7 : Real;
         rSpare8 : Real;
         tManCmd : Struct
            xSpare0 : Bool;   //
            xSpare1 : Bool;
            xSpare2 { ExternalWritable := 'False'} : Bool;
            xSpare3 { ExternalWritable := 'False'} : Bool;
            xSpare4 { ExternalWritable := 'False'} : Bool;
            xSpare5 { ExternalWritable := 'False'} : Bool;
            xSpare6 { ExternalWritable := 'False'} : Bool;
            xSpare7 { ExternalWritable := 'False'} : Bool;
            xSpare8 { ExternalWritable := 'False'} : Bool;
            xSpare9 { ExternalWritable := 'False'} : Bool;
            xSpare10 { ExternalWritable := 'False'} : Bool;
            xSpare11 { ExternalWritable := 'False'} : Bool;
            xSpare12 { ExternalWritable := 'False'} : Bool;
            xSpare13 { ExternalWritable := 'False'} : Bool;
            xSpare14 { ExternalWritable := 'False'} : Bool;
            xSpare15 { ExternalWritable := 'False'} : Bool;
            xSpare16 : Bool;
            xSpare17 : Bool;
            xSpare18 : Bool;
            xSpare19 : Bool;
            xSpare20 : Bool;
            xSpare21 : Bool;
            xSpare22 : Bool;
            xSpare23 : Bool;
            xSpare24 : Bool;
            xSpare25 : Bool;
            xSpare26 : Bool;
            xSpare27 : Bool;
            xSpare28 : Bool;
            xSpare29 : Bool;
            xSpare30 : Bool;
            xSpare31 : Bool;
         END_STRUCT;
      END_STRUCT;
   END_STRUCT;


BEGIN

END_DATA_BLOCK

